# B&R Automation Studio project PLC code - cp (part 13)

### Dryer.typ
```iecst
TYPE
	DryerModel_enum :
		(
		DryerNoType,
		DryerType_NOZ2_NIR_ARCLAMP,
		DryerType_NOZ2_NIR
		);
	DryerMachineStatus_enum :
		(
		DRYERMACH_STOPPED,
		DRYERMACH_PREPARINGTOMOVE,
		DRYERMACH_MOVING,
		DRYERMACH_PREPARING,
		DRYERMACH_PREPARED,
		DRYERMACH_STARTING,
		DRYERMACH_DRYING,
		DRYERMACH_STOPPING_DRYING,
		DRYERMACH_STOPPING_TRANSPORT,
		DRYERMACH_PREPARINGEMPTYBELT, (*Only vaccum transport on*)
		DRYERMACH_ERROR
		);
	Dryer_ProductDetectInputs : 	STRUCT
		pPDSignalSensorL1 : UDINT; (*Pointer to ProductDetect Signal coming directly from the sensor*)
		pPDSignalSensorL2 : UDINT; (*Pointer to ProductDetect Signal coming directly from the sensor*)
	END_STRUCT;
	Dryer_TempInputs : 	STRUCT
		iBoardInRaw : INT;
		iBoardOutRaw : INT;
		iBeltRaw : INT;
		iAirBlowerInputRaw : INT; (*45214336. -50C to +200C. 4-20mA*)
		iAirBlowerOutputRaw : INT; (*45214336. -50C to +200C. 4-20mA*)
		xBoardInSensorError : BOOL; (*Sensor Error*)
		xBoardOutSensorError : BOOL; (*Sensor Error*)
		xBeltSensorError : BOOL; (*Sensor Error*)
		xAirBlowerInputSensorError : BOOL; (*45214336. -50C to +200C. 4-20mA. Sensor Error*)
		xAirBlowerOutputSensorError : BOOL; (*45214336. -50C to +200C. 4-20mA. Sensor Error*)
	END_STRUCT;
	Dryer_InputsButtons : 	STRUCT
		xStopBlowers : BOOL;
		xManual : BOOL;
		xZero : BOOL;
		xAuto : BOOL;
		xStop : BOOL; (*EDGE*)
		xReset : BOOL;
	END_STRUCT;
	Dryer_SafetyInputs : 	STRUCT
		xMovementsEnabled : BOOL;
		xRemoteEStopOK : BOOL; (*Remote Emergency Stop*)
		xEStopFrontOK : BOOL;
		xEStopRearOK : BOOL;
		xClosedFrontInput : BOOL; (*Closed door detection*)
		xClosedFrontOutput : BOOL; (*Closed door detection*)
		xClosedRearInput : BOOL; (*Closed door detection*)
		xClosedRearOutput : BOOL; (*Closed door detection*)
	END_STRUCT;
	Dryer_Inputs : 	STRUCT
		Sw : Dryer_Inputs_Sw;
		Safety : Dryer_SafetyInputs;
		xStart : {REDUND_UNREPLICABLE} BOOL; (*EDGE*)
		xManual_GI : BOOL;
		xZero_GI : BOOL;
		xAuto_GI : BOOL;
		xMute : BOOL;
		xMain24VdcOK : BOOL;
		xFan24VdcOK : BOOL;
		xFanBreakersOK : BOOL;
		xFanBreakersWarning : BOOL; (*Power higher than 80% for all fans*)
		xConsentOk : BOOL;
		xExternalCleaningOrder : BOOL;
		iMachineModelCode : INT;
		xOpenDoorsKey : BOOL; (*Enable open doors with ArcLamp hot*)
		Temp : Dryer_TempInputs;
		ProductDetect : Dryer_ProductDetectInputs;
		Buttons : Dryer_InputsButtons;
	END_STRUCT;
	Dryer_HwData : 	STRUCT
		Family : USINT;
		Name : STRING[20];
		SerialNumber : STRING[80]; (*Serial number of the machine*)
	END_STRUCT;
	Dryer_Excutions : 	STRUCT
		slow : UDINT;
		fast : UDINT;
	END_STRUCT;
	Dryer_States_Position : 	STRUCT
		xGoingToPrint : BOOL; (*Internal bool used on printer to set state NOT CAP/NOT PRINT in printer*)
		xInPrint : BOOL; (*Internal bool used on printer to set state PRINTING in printer*)
		xCleaning : BOOL; (*Internal bool used on printer to set state CLEANING in printer*)
		xGoingToCap : BOOL; (*Internal bool used on printer to set state NOT CAP/NOT PRINT in printer*)
		xInCap : BOOL; (*Internal bool used on printer to set state CAPPED in printer*)
	END_STRUCT;
	Dryer_States_AutoLocation : 	STRUCT
		xLocalORManual : BOOL; (*Local settings and orders*)
		xLocal : BOOL; (*Local settings and orders*)
		xRemote : BOOL; (*Remote settings and orders*)
	END_STRUCT;
	Dryer_States_Mode : 	STRUCT
		xManual : {REDUND_UNREPLICABLE} BOOL; (*State to define Manual Mode*)
		xZero : BOOL; (*State to define Zero Mode*)
		xAuto : BOOL; (*State to define Auto Mode*)
		xStartUp : BOOL; (*State to define StartUp Mode*)
	END_STRUCT;
	Dryer_States_Out : 	STRUCT
		xOnline : BOOL;
		xError : BOOL;
		xDrying : BOOL;
		xDryerPresent : BOOL;
		xReadyToDry : BOOL;
		xJamDetection : BOOL;
		xTransportMoving : BOOL;
		xInRemote : BOOL;
		iModelVersion1 : UINT;
		iModelVersion2 : UINT;
		xMediaPresent : BOOL;
		xReadyToEmptyBelt : BOOL;
		xBeltEmpty : BOOL; (*Belt empty in the device*)
	END_STRUCT;
	Dryer_States_Temp : 	STRUCT
		rBoardIn : REAL;
		rBoardOut : REAL;
		rBelt : REAL;
		rAirBlowerInput : REAL;
		rAirBlowerOutput : REAL;
	END_STRUCT;
	Dryer_States_HMI : 	STRUCT
		xDryerLocalStopped : BOOL;
		xDryerStopped : BOOL;
		xShowThickness : BOOL; (*Thickness and Gap is used in the program and can be adjusted*)
		xVirtualMedia : BOOL;
		xShowEnableNIR : BOOL; (*Variable to let NIR enabling*)
	END_STRUCT;
	Dryer_States : 	STRUCT
		Position : Dryer_States_Position;
		Mode : Dryer_States_Mode;
		AutoLocation : Dryer_States_AutoLocation;
		LocationControl : MachineAutoLocation_enum;
		Out : Dryer_States_Out;
		DryerState : DryerMachineStatus_enum;
		Temp : Dryer_States_Temp;
		xConsent : BOOL; (*Internal bool used on printer to set state in CONSENT printer*)
		iAutoModeSW : INT; (*Printer State to sw *)
		iMachineModelCodeSW : INT; (*Printer model to Sw, in function of HW ID code*)
		xNotAutoPossible : BOOL; (*Some condition is preventing to entering auto*)
		StateMode : enumEFI_GenMachineState; (*states*)
		AutoMode : stEFI_MachineAutoModes; (*commands*)
		uiLicenseCounter : UINT;
		exec : Dryer_Excutions;
		HwData : Dryer_HwData;
		xAnyProductDetect : BOOL; (*Any product detect. In any line and coming from Carriage or Sensor directly. It means that a media has been printed*)
		xProductDetectL1 : BOOL; (*Any product detect in L1. In any line and coming from Carriage or Sensor directly. It means that a media has been printed*)
		xProductDetectL2 : BOOL; (*Any product detect in L2. In any line and coming from Carriage or Sensor directly. It means that a media has been printed*)
		xMediaDetected : BOOL; (*Media detected before product detect. Detected in Analog or in 3sensors*)
		iJamDevices : USINT := 0; (*Quantity of Jam Devices installed in the machine*)
		xStarted : BOOL; (*TRUE if the PLC is running*)
		HMI : Dryer_States_HMI;
	END_STRUCT;
	Dryer_ConstantParameters : 	STRUCT
		rMinThicknessMedia : REAL; (*mm*)
		rMaxThicknessMedia : REAL; (*mm*)
		rMountedMediaLevelInBypassMode : REAL; (*mm*)
		rMinMargin : REAL; (*mm*)
		rMaxMargin : REAL; (*mm*)
		rDistanceThicknesToPD : REAL; (*Distance Between Thicknes Detection To PD Sensor (mm)*)
		iNumBlocks : USINT; (*For writting the number of blocks in a machine*)
		iNumTransVacuum : USINT; (*For writting the number of TransportVacuum in a machine*)
		iNumJamModules : USINT; (*DEPRECATED!!. //TODELETE For writing the number of Jam Detection modules in a machine*)
		iNumSensorsPerJamDevice : USINT := 4; (*For writing the number of Sensors in each Jam Device*)
		rMaxBeltTorque : REAL := 25; (*Max torque supported by the Belt, independently of the motor itself in N·m*)
		rMaxBeltTempSlow : REAL := 180; (*Max temperature supported by the Belt during 30sec, in ºC*)
		rMaxBeltTempFast : REAL := 190; (*Max temperature supported by the Belt during 2sec, in ºC*)
	END_STRUCT;
	Dryer_CleanBeltParameters : 	STRUCT
		xCleanBeltContinue : BOOL; (*Input software parameter from Sw*)
		xCleanBeltByTiles : BOOL; (*Input software parameter from Sw*)
		xCleanBeltByTime : BOOL; (*Input sw param using time param iCleaningBeltByTime*)
		tiCleaningBeltDuration : TIME; (*Time in seconds. Input software parameter from Sw*)
		iCleaningBeltByTime : UINT; (*Time in Minutes. Input software parameter from Sw*)
		xCleanBeltForced : BOOL; (*Edge Command. Input software parameter from Sw*)
		iSPTilesToCleanBelt : UINT; (*Input software parameter from Sw*)
	END_STRUCT;
	Dryer_SuctionParameters : 	STRUCT
		iBlowerMode : INT; (*Suction mode functionality. It can be configured by GUI with Ventrui when is 1 or Turbine when is 2. Parameters received from GUI*)
		tiBlowerDelayOff : TIME; (*Delay time before turning off the turbine in auto mode*)
	END_STRUCT;
	Dryer_SafetyParameters : 	STRUCT
		rMarginSafePrint : REAL; (*SoftwareInput. Fix offset to bent tile. The heads go to the thickness measured + this value. Value in mm*)
		rMaxBeltSpeedSetPoint : REAL := 70.0; (*Max speed received from gui in m/min*)
	END_STRUCT;
	Dryer_DocumentParameters : 	STRUCT
		rWidth : REAL; (*Board's width in mm*)
		rLength : REAL; (*Board's length in mm*)
		rOffsetL1 : REAL;
		rOffsetL2 : REAL;
	END_STRUCT;
	Dryer_ThermalInertiaReduction : 	STRUCT
		iBoardsToStartReducing : USINT; (*Total boards detected to start reducing the power*)
		iBoardsToMaxPowerReduction : USINT; (*Total boards detected to form maximum power reduction*)
		rMaxPowerReduction : REAL; (*Maximum power reduction for thermal inertia*)
	END_STRUCT;
	Dryer_MediaParameters : 	STRUCT
		rThickness : REAL; (*Tile thickness to print from gui in mm*)
		rWidth : REAL; (*Board's width in mm*)
		rGap : REAL; (*Gap between boards in mm*)
		rLength : REAL; (*Board's length in mm*)
		rMargin : REAL; (*SoftwareInput, dry margin in mm*)
		rOffsetRegisterL1 : REAL;
	END_STRUCT;
	Dryer_SwParameters : 	STRUCT
		CleanBelt : Dryer_CleanBeltParameters;
		Suction : Dryer_SuctionParameters;
		Safety : Dryer_SafetyParameters;
		Media : stThicknessCtrl_MediaConfig;
		xDoubleLine : BOOL; (*0: Derecha 1: Izquierda*)
		xMachineDirection : BOOL; (*0: Derecha 1: Izquierda*)
		xEnableNir : BOOL;
		xEnableDDC : BOOL; (*Enable DDC in Dryer*)
		xEnableArcLamp : BOOL;
		rSubstratePowerReduction : REAL := 1.0; (*Substrate power reduction. From 1.0 (default) to 0.3 is allowed*)
		tiDelayConsent : TIME; (*Used on kernel to PLC. Time in seconds*)
		rBeltSpeedSetPoint : REAL := 20.0; (*Speed in m/min. Input parameter from SW*)
		xLineEmptyingBelt : BOOL; (*Line in emptying belt*)
		xPrinterBeltRuning : BOOL; (*Printer belt runing status*)
	END_STRUCT;
	Dryer_Parameters : 	STRUCT
		SW : Dryer_SwParameters; (*Software input params*)
		CT : Dryer_ConstantParameters; (*Printer input constants params*)
		ThermalInertia : Dryer_ThermalInertiaReduction;
		ConfigName : STRING[80];
		ConfigNameID : USINT := 0; (*Identification of the Configuration been executed*)
		xTransVacuumIndependenParams : BOOL; (*TRUE: Each TransVacuum with different parameters. FALSE: TransVacuum[1] copied to the rest of elements*)
		MachineModel : DryerModel_enum; (*HW ID codes are defined here*)
		PDSignalTpe : ProductDetectSignal_enum;
		xLeftHandMachine : BOOL; (*Software Output*)
		xRightHandMachine : BOOL; (*Software Output*)
		xLocalDisableDDC : BOOL;
		xEnableDryDocWidth : BOOL; (*Enable drying width by image instead of media, only in remote mode.*)
	END_STRUCT;
	Dryer_commands_Auto : 	STRUCT
		xPrepareToDry : BOOL;
		xStartDrying : BOOL;
		xRunTransport : BOOL;
		xPrepareToEmptyBelt : BOOL;
	END_STRUCT;
	Dryer_commands : 	STRUCT
		xAllToCap : BOOL; (*Use as EDGE*)
		xAllToPrint : BOOL; (*Use as EDGE*)
		xToLocal : BOOL; (*Command to go in Local mode*)
		xToRemote : BOOL; (*Command to go in Remote mode*)
		xResetSwitch : BOOL;
		xResetHub : BOOL;
		xResetFanBreaker : BOOL;
		xUnlockDoors : BOOL; (*Use as EDGE*)
		SerialNumber : stGeneral_SerialNumberCommands;
	END_STRUCT;
	Dryer_Inputs_Sw : 	STRUCT
		xStart_GI : BOOL; (*EDGE*)
		xStop_GI : BOOL; (*Edge command*)
		xMute_GI : BOOL; (*EDGE*)
		xPause_GI : BOOL; (*EDGE*)
		xReset_GI : BOOL; (*EDGE*)
		xToStop_GI : BOOL; (*Edge commandBool to Stop Mode*)
		xToNormal_GI : {REDUND_UNREPLICABLE} BOOL; (*Edge commandBool to start AutoRun Mode*)
		xToByPass_GI : BOOL; (*Edge commandBool to start Bypass Mode*)
		xStopBlowers_GI : BOOL; (*To stop blowers after keep them off to avoid cardboard fire*)
	END_STRUCT;
	Dryer_AutoCommands : 	STRUCT
		iAutoMode : enumEFI_MachineAutoStatesMode; (*Internal variable to manage AUTOMATIC modes in printer RU,BUPASS, LAB AND STOP*)
		xMuteAlarms : BOOL; (*Edge commandBool used to mute all alarms*)
		xToCap : BOOL; (*Edge commandBool used to send all block to cap*)
		xToPrint : BOOL; (*Edge commandBool used to send all block to print*)
		xReset : BOOL; (*Internal bool used on printer to set state RESET in printer*)
		xStart : BOOL; (*Edge Command to Start the Machine. By button or an specific order from Sw*)
		xStop : BOOL; (*Edge Command to Stop the Machine. By button or an specific order from Sw*)
	END_STRUCT;
	Dryer_AlarmsSafety : 	STRUCT
		xMaintenanceKey : BOOL; (*Maintenance Key active. Enables without safety guard closed*)
		xRemoteEStop : BOOL; (*Remote Emergency Stop*)
		xEStopFront : BOOL; (*Emergency Stop*)
		xEStopRear : BOOL; (*Emergency Stop*)
		xOpenedFrontInput : BOOL; (*Door*)
		xOpenedFrontOutput : BOOL; (*Door*)
		xOpenedRearInput : BOOL; (*Door*)
		xOpenedRearOutput : BOOL; (*Door*)
	END_STRUCT;
	Dryer_AlarmsList : 	STRUCT
		Safety : Dryer_AlarmsSafety;
		xAlarmPlarformInc : BOOL; (*AlarmCritical*)
		xAlarmComPcPLC : BOOL; (*AlarmStop*)
		xAlarmMountedMedia : BOOL;
		xAlarmMountedPieceBypassMode : BOOL; (*AlarmStop*)
		xUpNotConsent : BOOL; (*Resume alarms*)
		xNoActionDangerCollision : BOOL; (*Resume alarms*)
		xNoActionAlarmExist : BOOL; (*Resume alarms*)
		xPDBrokenSensorL1 : BOOL; (*Product Detect Line 1 Broken or Desconected*)
		xPDBrokenSensorL2 : BOOL; (*Product Detect Line 2 Broken or Desconected*)
		xMain24Vdc : BOOL; (*Main 24VDC Power Supply switched off*)
		xFan24Vdc : BOOL; (*Fan 24VDC Power Supply switched off*)
		xFanBreakers : BOOL; (*Fan breakers error*)
		xAlrBeltOvertorque : BOOL; (*Alarm Critical: Overtorque in Belt. Risk to break the belt itself*)
		xAlrBeltOverTempSlow : BOOL; (*Alarm Critical: OverTemperature in Belt. Risk to break the belt itself*)
		xAlrBeltOverTempFast : BOOL; (*Alarm Critical: OverTemperature in Belt. Risk to break the belt itself*)
		xAlrJam : BOOL; (*Alarm Critical: Any jam is triggered*)
		xAlrWrongPhysConf : BOOL; (*Alarm Critical: Wrong physical configuration or some tarjet are disconected*)
	END_STRUCT;
	Dryer_WarningsList : 	STRUCT
		xNotEnabledMovement : BOOL;
		xKeyMantenanceActive : BOOL; (*Key mantenance is active. No movements*)
		xValidConfiguration : BOOL; (*Review*)
		xMaxMovsBentTile : BOOL;
		xBentMedia : BOOL;
		xFanBreakersHighLoad : BOOL; (*Fan breakers High Load*)
		xMountedMediaInside : BOOL;
		xMediaStoppedInside : BOOL;
		xBoardInSensorError : BOOL; (*Sensor Error*)
		xBoardOutSensorError : BOOL; (*Sensor Error*)
		xBeltSensorError : BOOL; (*Sensor Error*)
		xAirBlowerInputSensorError : BOOL; (*45214336. -50C to +200C. 4-20mA. Sensor Error*)
		xAirBlowerOutputSensorError : BOOL; (*45214336. -50C to +200C. 4-20mA. Sensor Error*)
		xFrontDoorOpened : BOOL;
		xJamLowCrash : BOOL; (*Low level jam detected by the jam device*)
		xRearDoorOpened : BOOL;
	END_STRUCT;
	Dryer_Alarms : 	STRUCT
		Warning : Dryer_WarningsList;
		Alarm : Dryer_AlarmsList;
		xAlrStopDrying : BOOL;
		iReasonStopDrying : UINT;
		xAlrDisableGoToProduction : BOOL;
		xAlrSafetySystemEStop : BOOL; (*SLX DI 10 is enable transport from safety progam*)
		xAlarmSound : BOOL;
	END_STRUCT;
	Dryer_Log : 	STRUCT
		ManualChg : DINT;
		AutoChg : DINT;
		ManualHrs : DINT;
		AutoHrs : DINT;
		VdcHrs : DINT;
		DateStart : DINT;
		iPieceCounterBtwCleaningsL2 : INT;
		iPieceCounterBtwCleaningsL1 : INT;
		udiBentTilesCounter : UDINT;
		udiPiecesCounterErrorL1 : UDINT; (*PD Detection Counter Failed L1*)
		udiPiecesCounterErrorL2 : UDINT; (*PD Detection Counter Failed L2*)
		udiPiecesCounterL1 : UDINT;
		udiPiecesCounterL2 : UDINT;
		udiTileCounterBalluffLaser : UDINT; (*Program in mode active..end*)
		udiTileCounterTriggerLaser : UDINT; (*Program in mode active..end*)
		udiDifCounters : UDINT; (*Program in mode active..end*)
		iTilesCounterToClean : UINT;
	END_STRUCT;
	Dryer_Outputs : 	STRUCT
		xResetSwitch : BOOL;
		xResetHub : BOOL;
		xResetFanBreaker : BOOL;
		xLockFrontDoor : BOOL;
		xLockRearDoor : BOOL;
		xBuzzer : BOOL;
		xRedLight : BOOL;
		xYellowLight : BOOL;
		xBlueLight : BOOL;
		xWhiteLight : BOOL;
		xResetBlueLight : BOOL;
		xConsentL1 : BOOL;
		xConsentL2 : BOOL;
		xSuctionTurbine : BOOL;
		xLightReset : BOOL;
		xCoolingPCStart : BOOL;
		xKeepSafetyNIR : BOOL;
	END_STRUCT;
	DryerMachine : 	STRUCT
		In : Dryer_Inputs;
		St : Dryer_States;
		Pt : Dryer_Parameters;
		commands : Dryer_commands;
		AutoCmd : Dryer_AutoCommands;
		AlSummary : stEFI_AlarmSummary;
		Al : Dryer_Alarms;
		Lg : Dryer_Log;
		Out : Dryer_Outputs;
	END_STRUCT;
	DryerRemoteSignals : 	STRUCT
		xMediaPresent : BOOL; (*Media present at the entrance of the machine*)
		xBreakerOKBlowerInput : BOOL;
		xBreakerOKBlowerOutput : BOOL;
		Safety : Dryer_SafetyInputs;
	END_STRUCT;
	DryerRemoteData : 	STRUCT
		xCommsOK : BOOL; (*The comunications are working fine. Data can be trusted*)
		Parameters : Dryer_SwParameters;
		Commands : Dryer_commands_Auto; (*From Line to Dryer*)
		Signals : DryerRemoteSignals;
	END_STRUCT;
END_TYPE
```

### InksBox.typ
```iecst
TYPE
	InkboxCabinetParameters : 	STRUCT
		MaxTempPowerPsu : UINT; (*Power in Watts*)
		TotalInksPerPsu : USINT;
		TotalInkSystems : USINT;
	END_STRUCT;
	InkboxParameters : 	STRUCT
		TotalCabinets : USINT;
		Cabinets : ARRAY[0..MAX_LAST_INK_CABINET]OF InkboxCabinetParameters;
	END_STRUCT;
	InkboxCabinetStatus : 	STRUCT
		xExists : BOOL; (*The cabinet exists*)
		rPowerReduction : REAL; (*Power reduction calculated*)
		rTotalAskedPower : REAL; (*The total power calculated by the Inks*)
	END_STRUCT;
	InkboxCommands : 	STRUCT  (*Just Edge commands*)
		xReset : BOOL;
		xMute : BOOL;
	END_STRUCT;
	InkboxStatus : 	STRUCT
		iTotalInks : USINT; (*Total possible Inks by cabinets configuration*)
		ExistingInks : ARRAY[0..MAX_LAST_INK]OF BOOL;
		Cabinets : ARRAY[0..MAX_LAST_INK_CABINET]OF InkboxCabinetStatus;
	END_STRUCT;
	InkBox : 	STRUCT
		Status : InkboxStatus;
		Parameters : InkboxParameters;
		Commands : InkboxCommands; (*Just Edge Commands*)
	END_STRUCT;
END_TYPE
```

### Global.var
```iecst
VAR
	iIndexWhiteCuringLedBar : USINT;
	iIndexColorCuringLedBar : USINT;
	iIndexPrimerCuringLedBar : USINT;
	gSafetyController : stSafetyController;
	gBelt : stBelt;
	gBeltClean : BeltClean_typ;
	gBlock : ARRAY[0..MAX_LAST_BLOCK] OF StBlock; (*Logical array of Blocks in the machine. Starts in 0 because it is used in a C program*)
	gSimpleBlock : ARRAY[0..MAX_LAST_SIMPLEBLOCK] OF SimpleBlock; (*Logical array of Blocks in the machine. Starts in 0 because it is used in a C program*)
	gBlockInputs : ARRAY[0..MAX_LAST_BLOCK] OF StBlock_Inputs; (*Used for mapping physical inputs block to logical block*)
	gBlockOutputs : ARRAY[0..MAX_LAST_BLOCK] OF StBlock_Outputs; (*Used for mapping physical outputs block to logical block*)
	gPowermeters : ARRAY[0..2] OF stPowerMeter;
	gChiller : ARRAY[0..MAX_LAST_CHILLER] OF StChiller; (*Struct for chiller configuration*)
	gPlcDiagMC_Pt : StGeneral_Parameters;
	gTransVacuum : ARRAY[0..MAX_LAST_TRANS_VACUUM] OF TransVacuum_typ;
	gNonCrash : ARRAY[0..MAX_LAST_NON_CRASH] OF NonCrash_typ;
	gCuringLed : ARRAY[0..MAX_LAST_CURING_LED] OF CuringLed_typ;
	gDing : stThicknessAnalog_typ;
	gOverVarnish : Opv_typ;
	gPrimer : Primer_typ;
	gStacker : Stacker_typ;
	gDryerAnc : DryerAnc_typ;
	gLine : LineControl_typ;
	gEventLogLoader : EventLoader;
	gEventLogManager : EventManager;
	gInks : ARRAY[0..MAX_LAST_INK] OF stInks; (*Logical array of InkSystems in the machine. Starts in 0 because it is used in a C program*)
	gInksConstants : stInksConstantsToSw; (*horrible!! Pending to change *)
	gSarm : Sarm_typ;
	gFeeder : Feeder_typ;
	gInksInputs : ARRAY[0..MAX_LAST_INK] OF stInksSignalsIn; (*0 is not used. Just to compile in C*)
	gInksOutputs : ARRAY[0..MAX_LAST_INK] OF stInksSignalsOut;
	gJamInputs : ARRAY[0..MAX_LAST_JAMDEVICE] OF JamDetectInputs_typ;
	gJamOutputs : ARRAY[0..MAX_LAST_JAMDEVICE] OF JamDetectOutputs_typ;
	gMachine : StGeneral;
	gDryer : DryerMachine;
	gNirAdphos : NIRAdphos;
	gPairedMotors : ARRAY[0..2] OF PairedIclaMotors_typ; (*Paired icla motors structure*)
	gEdgeHoldDown : EdgeHoldDown_typ; (*Edge hold down structure*)
	gPhotoCells : nSensors_typ; (*gPhotocells structure*)
	gPLC : StPLC;
	gThicknessCtrl : stThicknessCtrl_typ;
	gBasicDetectMedia : DetectionMedia;
	gArcLampGew : ArcLampGew;
	g_xInputSelectMachine : BOOL;
	gJamDetect : ARRAY[0..MAX_LAST_JAMDEVICE] OF JamDetect_typ;
	gAirCleaner : StGeneral_AirCleaner;
	gCamera : StGeneral_Camera;
	gJamCamera : JamPerBar_typ;
	gJamPerCuringLed : ARRAY[0..MAX_LAST_CURING_LED] OF JamPerBar_typ;
	gJamPerInk : ARRAY[0..MAX_LAST_INK] OF JamPerBar_typ;
	gInkBox : InkBox;
	gTime : TimeMachine;
	gInverterSignalsPowerLink : ARRAY[0..MAX_LAST_INVERTER] OF AxisP66_Signals_typ;
	gInverterSignalsCanOpen : ARRAY[0..MAX_LAST_INVERTER] OF AxisP66_Signals_typ;
	gInverterSignalsPowerLinkABB : ARRAY[0..MAX_LAST_INVERTER] OF AxisP66_Signals_typ;
	gPlcCards : ARRAY[0..100] OF PLCCardData;
	xShowSecondLayout : BOOL := FALSE; (*Show second card block layout in diagnostic screen*)
	xShowThirdLayout : BOOL := FALSE; (*Show third card block layout in diagnostic screen*)
	stConfigToShow_Lyout1 : STRING[80] := 'P4_PDC_content'; (* Configuration ID to show in HMI || P4_PDC_content ; SHIELD_Cards_content ; NZ2_Cards_content*)
	stConfigToShow_Lyout2 : STRING[80] := 'P4_block1_content'; (*Configuration ID to show in HMI || P4_block1_content ; NZ2_Printer_content*)
	stConfigToShow_Lyout3 : STRING[80] := 'P4_block2_content'; (*Configuration ID to show in HMI || P4_block2_content*)
END_VAR
```

### Global_IO.var
```iecst
VAR
	X20CPUData : PlcCardMapping; (*Map: P4&EBRO*)
	X1 : PlcCardMapping; (*Map: P4&EBRO*)
	X2 : PlcCardMapping; (*Map: P4&EBRO*)
	X3 : PlcCardMapping; (*Map: P4&EBRO*)
	X20DOF322_001 : PlcCardMapping; (*Map: P4*)
	X20DIF371_001 : PlcCardMapping; (*Map: EBRO&S1400*)
	X20DIF371_002 : PlcCardMapping; (*Map: P4&EBRO&S1400*)
	X20DIF371_003 : PlcCardMapping; (*Map: P4&EBRO$S1400*)
	X20DOF322_004 : PlcCardMapping; (*Map: P4*)
	X20DIF371_004 : PlcCardMapping; (*Map: EBRO*)
	X20DIF371_005 : PlcCardMapping; (*Map: S1400*)
	X20DIF371_006 : PlcCardMapping; (*Map: S1400*)
	X20AI2636_005 : PlcCardMapping; (*Map: P4*)
	X20DOF322_005 : PlcCardMapping; (*Map: EBRO*)
	X20SLX402_006 : PlcCardMapping; (*	X20SI2100_010 : PlcCardMapping; Map: P4*)
	X20DOF322_006 : PlcCardMapping; (*Map: EBRO*)
	X20AI4322_008 : PlcCardMapping; (*Map: EBRO*)
	X20AI4322_102 : PlcCardMapping; (*Map: InkBox*)
	X20AI4322_202 : PlcCardMapping; (*Map: InkBox*)
	X20AI4322_302 : PlcCardMapping; (*Map: InkBox*)
	X20AT2222_103 : PlcCardMapping; (*Map: InkBox*)
	X20AT2222_203 : PlcCardMapping; (*Map: InkBox*)
	X20AT2222_303 : PlcCardMapping; (*Map: InkBox*)
	X20DOF322_104 : PlcCardMapping; (*Map: InkBox*)
	X20DOF322_204 : PlcCardMapping; (*Map: InkBox*)
	X20DOF322_304 : PlcCardMapping; (*Map: InkBox*)
	X20AO4622_105 : PlcCardMapping; (*Map: InkBox*)
	X20AO4622_205 : PlcCardMapping; (*Map: InkBox*)
	X20AO4622_305 : PlcCardMapping; (*Map: InkBox*)
	X20DI9372_008 : PlcCardMapping; (*Map: S1400*)
	X20AO4622_009 : PlcCardMapping; (*Map: EBRO*)
	X20DOF322_009 : PlcCardMapping; (*Map:S1400*)
	X20DOF322_010 : PlcCardMapping; (*Map:S1400*)
	X20AT4222_010 : PlcCardMapping; (*Map: EBRO*)
	X20DOF322_011 : PlcCardMapping; (*Map:S1400*)
	X20DOF322_012 : PlcCardMapping; (*Map:S1400*)
	X20DOF322_013 : PlcCardMapping; (*Map:S1400*)
	X20AI8321_015 : PlcCardMapping; (*Map:S1400*)
	X20AI8321_016 : PlcCardMapping; (*Map:S1400*)
	X20AI8321_111 : PlcCardMapping; (*Map:S1400*)
	X20AI8321_112 : PlcCardMapping; (*Map:S1400*)
	X20AI8321_113 : PlcCardMapping; (*Map:S1400*)
	X20AI8321_114 : PlcCardMapping; (*Map:S1400*)
	X20AI8321_018 : PlcCardMapping; (*Map:S1400*)
	X20AI8321_019 : PlcCardMapping; (*Map:S1400*)
	X20AO4622_017 : PlcCardMapping; (*Map:S1400*)
	X20AO4622_018 : PlcCardMapping; (*Map:S1400*)
	X20AO4622_019 : PlcCardMapping; (*Map:S1400*)
	X20AO4622_020 : PlcCardMapping; (*Map:S1400*)
	X20AT4222_022 : PlcCardMapping; (*Map:S1400*)
	X20AT4222_023 : PlcCardMapping; (*Map:S1400*)
	X20AI2636_024 : PlcCardMapping; (*Map:S1400*)
	X20AI8321_025 : PlcCardMapping;
	X20AI8321_024 : PlcCardMapping;
	X20DIF371_024 : PlcCardMapping; (*Map:S1400*)
	X20AI8321_026 : PlcCardMapping; (*Map:S1400*)
	X20AT4222_027 : PlcCardMapping;
	X20AT4222_028 : PlcCardMapping;
	X20AT4222_029 : PlcCardMapping; (*Map:S1400*)
	X20AT4222_030 : PlcCardMapping; (*Map:S1400*)
	X20DIF371_030 : PlcCardMapping; (*Map: P4*)
	X20AI2636_100 : PlcCardMapping;
	X20DIF371_101 : PlcCardMapping; (*Map: P4 & Map: InkBox*)
	X20DIF371_102 : PlcCardMapping; (*Map: P4*)
	X20DIF371_103 : PlcCardMapping; (*Map: P4*)
	X20DIF371_104 : PlcCardMapping; (*Map: P4*)
	X20DIF371_105 : PlcCardMapping; (*Map: P4*)
	X20DIF371_106 : PlcCardMapping; (*Map: P4*)
	X20DI9372_107 : PlcCardMapping; (*Map: P4*)
	X20DIF371_107 : PlcCardMapping; (*Map: P4*)
	X20DC4395_104 : PlcCardMapping; (*Map: P4*)
	X20DC4395_105 : PlcCardMapping; (*Map: P4*)
	X20DOF322_106 : PlcCardMapping; (*Map: P4*)
	X20DOF322_107 : PlcCardMapping; (*Map: P4*)
	X20DOF322_108 : PlcCardMapping; (*Map: P4*)
	X20DOF322_109 : PlcCardMapping; (*Map: P4*)
	X20DOF322_110 : PlcCardMapping; (*Map: P4*)
	X20AI8321_109 : PlcCardMapping; (*Map: P4*)
	X20AI8321_110 : PlcCardMapping; (*Map: P4*)
	X20AO4622_111 : PlcCardMapping; (*Map: P4*)
	X20AO4622_112 : PlcCardMapping; (*Map: P4*)
	X20AO4622_113 : PlcCardMapping; (*Map: P4*)
	X20AO4622_114 : PlcCardMapping; (*Map: P4*)
	X20AO4622_115 : PlcCardMapping; (*Map: P4*)
	X20AO4622_116 : PlcCardMapping; (*Map: P4*)
	X20AO4622_117 : PlcCardMapping; (*Map: P4*)
	X20AT4222_114 : PlcCardMapping; (*Map: P4*)
	X20AT4222_115 : PlcCardMapping; (*Map: P4*)
	X20AT4222_116 : PlcCardMapping; (*Map: P4*)
	X20AT4222_117 : PlcCardMapping; (*Map: P4*)
	X20AT4222_118 : PlcCardMapping; (*Map: P4*)
	X20AT4222_119 : PlcCardMapping; (*Map: P4*)
	X20AT4222_120 : PlcCardMapping; (*Map: P4*)
	X20AT4222_121 : PlcCardMapping; (*Map: P4*)
	X20CS1030_150 : PlcCardMapping; (*Map: P4*)
	X20CS1030_151 : PlcCardMapping; (*Map: P4*)
	X20CS1030_121 : PlcCardMapping; (*Map: P4*)
	X20CS1030_180 : PlcCardMapping; (*Map: P4*)
	X20CS1030_181 : PlcCardMapping; (*Map: P4*)
	X20CS1030_162 : PlcCardMapping; (*Map: P4*)
	X20PS3300_114 : PlcCardMapping; (*Map: P4*)
	Pdc_X20DOF322_024 : PlcCardMapping;
	Pdc_X20DOF322_025 : PlcCardMapping;
	Pdc_X20DIF371_023 : PlcCardMapping;
	X20PS3300_106 : PlcCardMapping; (*Map: P4*)
	X20PS3300_020 : PlcCardMapping;
	X20PS3300_008 : PlcCardMapping;
	X20PS3300_157 : PlcCardMapping;
	X20PS3300_150 : PlcCardMapping;
	X20PS3300_115 : PlcCardMapping;
	X20PS3300_107 : PlcCardMapping;
	X20PS3300_152 : PlcCardMapping; (*Map: P4*)
	X20DIF371_151 : PlcCardMapping; (*Map: P4*)
	X20DIF371_152 : PlcCardMapping; (*Map: P4*)
	X20DIF371_153 : PlcCardMapping; (*Map: P4*)
	X20DIF371_154 : PlcCardMapping; (*Map: P4*)
	X20DOF322_155 : PlcCardMapping; (*Map: P4*)
	X20DOF322_156 : PlcCardMapping; (*Map: P4*)
	X20AI8221_156 : PlcCardMapping; (*Map: P4*)
	X20AO4622_157 : PlcCardMapping; (*Map: P4*)
	X20AO4622_158 : PlcCardMapping; (*Map: P4*)
	X20AO4622_159 : PlcCardMapping; (*Map: P4*)
	X20AO4622_160 : PlcCardMapping; (*Map: P4*)
	X20AO4622_161 : PlcCardMapping; (*Map: P4*)
	X20SI8110_117 : PlcCardMapping; (*Map: P4*)
	X20SO2110_118 : PlcCardMapping; (*Map: P4*)
	X20DIF371_201 : PlcCardMapping; (*Map: P4 & InkBox*)
	X20DIF371_202 : PlcCardMapping; (*Map: P4*)
	X20DIF371_203 : PlcCardMapping; (*Map: P4*)
	X20DIF371_301 : PlcCardMapping; (*Map: InkBox*)
	X20DC4395_204 : PlcCardMapping; (*Map: P4*)
	X20DC4395_205 : PlcCardMapping; (*Map: P4*)
	X20DIF371_180 : PlcCardMapping; (*Map: P4*)
	X20AI8321_181 : PlcCardMapping; (*Map: P4*)
	X20DOF322_205 : PlcCardMapping; (*Map: Dryer*)
	X20DOF322_206 : PlcCardMapping; (*Map: P4*)
	X20DOF322_207 : PlcCardMapping; (*Map: P4*)
	X20DOF322_208 : PlcCardMapping; (*Map: P4*)
	X20AI8321_207 : PlcCardMapping; (*Map: P4*)
	X20AI8321_209 : PlcCardMapping; (*Map: P4*)
	X20AI8321_210 : PlcCardMapping; (*Map: P4*)
	X20AO4622_208 : PlcCardMapping; (*Map: Dryer*)
	X20AO4622_211 : PlcCardMapping; (*Map: P4*)
	X20AO4622_212 : PlcCardMapping; (*Map: P4*)
	X20AO4622_213 : PlcCardMapping; (*Map: P4*)
	X20AT4222_209 : PlcCardMapping; (*Map: Dryer*)
	X20AT4222_214 : PlcCardMapping; (*Map: P4*)
	X20AT4222_215 : PlcCardMapping; (*Map: P4*)
	X20AT4222_216 : PlcCardMapping; (*Map: P4*)
	X20SI8110_217 : PlcCardMapping; (*Map: P4*)
	X20SO2110_218 : PlcCardMapping; (*Map: P4*)
	Reserve01 : PlcCardMapping;
	SiUnitBK1 : StSiUnit;
	SiUnitBK2 : StSiUnit;
	SiUnitPwrLnkBK1 : StSiUnitPwrLnk;
	Pdc_X20DIF371_001 : PlcCardMapping;
	Pdc_X20DIF371_002 : PlcCardMapping;
	Pdc_X20DIF371_003 : PlcCardMapping;
	Pdc_X20DIF371_004 : PlcCardMapping;
	Pdc_X20DIF371_005 : PlcCardMapping;
	Pdc_X20DIF371_006 : PlcCardMapping;
	Pdc_X20DIF371_007 : PlcCardMapping;
	Pdc_X20DIF371_009 : PlcCardMapping;
	Pdc_X20DIF371_030 : PlcCardMapping;
	Pdc_X20AI2636_050 : PlcCardMapping;
	Pdc_X20DIF371_060 : PlcCardMapping;
	Pdc_X20DIF371_070 : PlcCardMapping;
	X20PS3300_007 : PlcCardMapping;
	Pdc_X20DIF371_024 : PlcCardMapping;
	Pdc_X20DIF371_022 : PlcCardMapping;
	Pdc_X20DIF371_020 : PlcCardMapping;
	Pdc_X20DIF371_021 : PlcCardMapping;
	X20PS3300_006 : PlcCardMapping;
	X20PS3300_022 : PlcCardMapping;
	Pdc_X20DOF322_023 : PlcCardMapping;
	Pdc_X20DIF371_1 : PlcCardMapping;
	Pdc_X20DIF371_2 : PlcCardMapping;
	Pdc_X20DIF371_3 : PlcCardMapping;
	Pdc_X20DOF322_008 : PlcCardMapping;
	Pdc_X20DOF322_009 : PlcCardMapping;
	Pdc_X20DOF322_010 : PlcCardMapping;
	Pdc_X20DOF322_1 : PlcCardMapping;
	Pdc_X20DIF371_050 : PlcCardMapping;
	Pdc_X20DIF371_040 : PlcCardMapping;
	Pdc_X20DOF322_051 : PlcCardMapping;
	Pdc_X20DOF322_011 : PlcCardMapping;
	Pdc_X20DOF322_007 : PlcCardMapping;
	Pdc_X20DOF322_005 : PlcCardMapping;
	X20AO4622_119 : PlcCardMapping;
	X20AO4622_118 : PlcCardMapping;
	X20IF1072_SS1 : PlcCardMapping;
	X20IF1072_SS2 : PlcCardMapping;
	X20IF1072_SS3 : PlcCardMapping;
	X20SM1436_007 : PlcCardMapping;
	X20SM1436_008 : PlcCardMapping;
	X20SM1436_011 : PlcCardMapping;
	X20SM1436_012 : PlcCardMapping;
	X20SM1436_111 : PlcCardMapping;
	X20SM1436_112 : PlcCardMapping;
	X20PS3300_014 : PlcCardMapping;
	X20PS3300_021 : PlcCardMapping;
	X20BC0083 : PlcCardMapping;
	X20PS9400 : PlcCardMapping;
	FakeBoolInput : BOOL;
END_VAR
```

### GlobalComms.var
```iecst
VAR
	gToWriteDataModbSarm : ARRAY[1..25] OF UINT;
	gReceivedDataModbSarm : ARRAY[1..25] OF UINT;
	gToWriteDataModbFeeder : ARRAY[1..25] OF UINT;
	gReceivedDataModbFeeder : ARRAY[1..25] OF UINT;
	gToWriteDataModbStacker : ARRAY[1..25] OF UINT;
	gReceivedDataModbStacker : ARRAY[1..25] OF UINT;
	gToWriteDataModbOpv : ARRAY[1..25] OF UINT;
	gReceivedDataModbOpv : ARRAY[1..25] OF UINT;
	gToWriteDataModbPrimer : ARRAY[1..25] OF UINT;
	gReceivedDataModbPrimer : ARRAY[1..25] OF UINT;
	gToWriteDataModbTransport : ARRAY[1..25] OF INT;
	gReceivedDataModbTransport : ARRAY[1..25] OF INT;
	gReceivedDataModPowerMeter1 : ARRAY[0..120] OF UINT;
	gReceivedDataModPowerMeter2 : ARRAY[0..120] OF UINT;
	gReceivedDataModbSafety : ARRAY[0..20] OF UINT; (*0 Not used. Needed because used in the Tests*)
	gDryerRemoteData : DryerRemoteData; (*This is the data from the Printer to the Dryer*)
	gDryerLocalData : DryerInputs_typ; (*This is the data from the Dryer to the Printer*)
END_VAR
```

### MotionBasis.var
```iecst
(********************************************************************
 * COPYRIGHT - B&R Spain
 ********************************************************************
 * Package: MotionBasis
 * File: MotionBasis.var
 * Author: jorgemur
 * Created: September 19, 2018
 ********************************************************************
 * Variables of Motion
 ********************************************************************)
VAR
	gAxis : ARRAY[0..8] OF AxisCtrl_typ; (*Axis control structure. 1.Belt,2.Bk1,3.Bk2,4.SM1,5.SM2,6.NonCrash1,7.NonCrash28.Bk3*)
END_VAR
VAR RETAIN
	gAxisPermanEncData : ARRAY[0..8] OF MC_ENDLESS_POSITION; (*Permanent variable where encoder data is stored*) (*	gPermanentEncData2 : MC_ENDLESS_POSITION; *) (*Permanent variable where encoder data is stored*)
END_VAR
VAR
	gIcla : ARRAY[0..MAX_LAST_ICLA_MOTOR] OF stIcla; (*Physical array of Icla. index1>>Icla_A index2>>Icla_B*)
	gIclaNetData : ARRAY[0..MAX_LAST_ICLA_MOTOR] OF IclaNetData_typ; (*Physical array of IclaNetData. index1>>Icla_A index2>>Icla_B*)
	gAxisInverter : ARRAY[0..MAX_LAST_INVERTER] OF AxisP66_typ; (*Axis of the Inverters of the system of the family P66 & P67*)
END_VAR
VAR RETAIN
	gISQRippleData : ARRAY[0..8] OF MC_ISQ_RippleData_typ;
END_VAR
(* ********************************************************************
 * Identification of the Axis
 *******************************************************************
 #1. Belt
 #2. Vertical Block 1
 #3. Vertical Block 2
 #4. StepperMotor1 (3 Sensors)
 #5. StepperMotor2 (3 Sensors)
 #6. NonCrash 1
 #7. NonCrash 2
 #8. Vertical Block 3
 ********************************************************************)
```

### Simulation.var
```iecst
VAR
	gSimMachine : SimMachine_typ;
	gSimChiller : ARRAY[0..MAX_LAST_CHILLER] OF stChillerSim;
	gSimBlock : ARRAY[0..MAX_LAST_BLOCK] OF SimBlock_typ;
	gSimSimpleBlock : ARRAY[0..MAX_LAST_SIMPLEBLOCK] OF SimBlock_typ;
	gSimSarm : Sarm_typ;
	gSimFeeder : FeederSim_typ;
	gSimDryerAnc : DryerSimAnc_typ;
	gSimOverVarnish : PrimerSim_typ;
	gSimPrimer : PrimerSim_typ;
	gSimStacker : StackerSim_typ;
	gSimJamDetect : ARRAY[0..MAX_LAST_JAMDEVICE] OF JamDetectSim_typ;
	gSimInks : ARRAY[0..MAX_LAST_INK] OF SimInk_typ;
	gSimSafetyController : SafetyControllerSim_typ;
	gSimArcLamp : ArcLampSim_typ;
	gSimNirAdphos : NirAdphosSim_typ;
	gSimNonCrash : ARRAY[0..MAX_LAST_NON_CRASH] OF SimNonCrash_typ;
	gSimThickCtrl : SimThickCtrl_typ;
	gTestsExec : TestExecution;
	gSimDryer : SimDryer_typ;
END_VAR
```

### Program Logical/InkBox/Config/Initialize (IEC)

#### Initialize.st - Cyclic code
```iecst
PROGRAM _INIT

	HWInfoCpu.pName := ADR(gMachine.St.HwData.Name);
	HWInfoCpu.first := TRUE;
	HWInfoCpu.enable := TRUE;
	HWInfoCpu();
	gMachine.St.HwData.Family := HWInfoCpu.family;

	// Tranfer permanent vars when PLC is starting
	gMachine.parSw:= gPermanentMachine;

	FOR iInksIndex:=1 TO MAX_LAST_INK DO
		gInks[iInksIndex].parSw := gPermanentInksParSw[iInksIndex];
		gInks[iInksIndex].parameters.parBar := gInksPermanentParBar[iInksIndex];
	END_FOR

	gInkBox.Parameters := gPermanentInkBox;
	gBelt.parSw := gPermanentSwBelt;
	gTransVacuum[1].parSw := gPermanentTrVacuum[1];

END_PROGRAM

PROGRAM _CYCLIC

	//Assign the ConfigurationID been executed
	projectInfo(Execute:=gMachine.Pt.ConfigNameID=0); //Just to execute if still the configuration has not been read
	IF projectInfo.Done AND NOT projectInfo.Error THEN
		IF brsstrcmp(ADR(GC_CONFIG_INKBOX),ADR(projectInfo.ConfigurationID))=0 THEN

			IF gMachine.In.x230V THEN //This var is assigned to a ModuleOk just for simulation. Never in a real cabinet
				gMachine.Pt.ConfigNameID:=GC_CONFIG_INKBOX_SIM_ID;
			ELSE
				gMachine.Pt.ConfigNameID:=GC_CONFIG_INKBOX_ID;
			END_IF
		ELSE
			gMachine.Pt.ConfigNameID:=0;
		END_IF
		strcpy(ADR(gMachine.Pt.ConfigName),ADR(projectInfo.ConfigurationID));
	END_IF

END_PROGRAM
```

### Program Logical/InkBox/Config/SavePermanent

#### SavePermanent.st
```iecst
PROGRAM _CYCLIC

	// Permanents Vars
	gPermanentMachine:=gMachine.parSw;

	FOR iInksIndex:=1 TO MAX_LAST_INK DO
		gPermanentInksParSw[iInksIndex] := gInks[iInksIndex].parSw;
		gInksPermanentParBar[iInksIndex] := gInks[iInksIndex].parameters.parBar;
	END_FOR

	gPermanentInkBox := gInkBox.Parameters;
	gPermanentSwBelt := gBelt.parSw;
	gPermanentTrVacuum[1] := gTransVacuum[1].parSw;

	gPermanentVersion.iVersion0 := gPLC.iVersion0;
	gPermanentVersion.iVersion1 := gPLC.iVersion1;
	gPermanentVersion.iVersion2 := gPLC.iVersion2;
	gPermanentVersion.iVersion3 := gPLC.iVersion3;

END_PROGRAM
```

### Program Logical/InkBox/InkBoxCtrl/MainInkBox (IEC)

#### InternalPLC.st - Internal PLC Vars
```iecst
ACTION InternalPLC:

	// PLC VARS
	IF gPLC.diCycleTime =0 THEN
		gPLC.Internal.RestartInfo(enable := TRUE);
		gPLC.diCycleTime:=gPLC.Internal.RestartInfo.cycle_time;  // Is a fix cycle time

		gPLC.xColdRestart:= gPLC.Internal.RestartInfo.init_reason=1;
		gPLC.xWarmRestart:= gPLC.Internal.RestartInfo.init_reason=2;
		gPLC.xDownloadRestart:= gPLC.Internal.RestartInfo.init_reason=3;

		gPLC.xFirst_Scan :=	gPLC.Internal.RestartInfo.init_reason=-1 OR gPLC.xColdRestart OR gPLC.xWarmRestart OR gPLC.xDownloadRestart;

		gPLC.Internal.RestartInfo(enable := FALSE);

	ELSIF gPLC.xFirst_Scan THEN
		gPLC.xFirst_Scan:= FALSE;
		gPLC.xColdRestart:= FALSE;
		gPLC.xWarmRestart:= FALSE;
		gPLC.xDownloadRestart:= FALSE;
	END_IF

	//BLINK
	gPLC.Internal.Blink_100ms.T_Blink:=T#100MS;
	gPLC.Internal.Blink_100ms();
	gPLC.xBlk_100ms:= gPLC.Internal.Blink_100ms.Out;

	gPLC.Internal.Blink_200ms.T_Blink:=T#200MS;
	gPLC.Internal.Blink_200ms();
	gPLC.xBlk_200ms:= gPLC.Internal.Blink_200ms.Out;

	gPLC.Internal.Blink_500ms.T_Blink:=T#500MS;
	gPLC.Internal.Blink_500ms();
	gPLC.xBlk_500ms:= gPLC.Internal.Blink_500ms.Out;

	gPLC.Internal.Blink_1s.T_Blink:=T#1S;
	gPLC.Internal.Blink_1s();
	gPLC.xBlk_1s:= gPLC.Internal.Blink_1s.Out;

	gPLC.Internal.Blink_2s.T_Blink:=T#2S;
	gPLC.Internal.Blink_2s();
	gPLC.xBlk_2s:= gPLC.Internal.Blink_2s.Out;

	gPLC.Internal.Blink_5s.T_Blink:=T#5S;
	gPLC.Internal.Blink_5s();
	gPLC.xBlk_5s:= gPLC.Internal.Blink_5s.Out;

	gPLC.Internal.Blink_10s.T_Blink:=T#10S;
	gPLC.Internal.Blink_10s();
	gPLC.xBlk_10s:= gPLC.Internal.Blink_10s.Out;

	// License counter	and  Keep alive
	IF EDGEPOS(gPLC.xBlk_1s) THEN
		gMachine.St.uiLicenseCounter:= gMachine.St.uiLicenseCounter+1;
		gMachine.St.iFaultRunPlc:= gMachine.St.iFaultRunPlc+1;
	END_IF;

END_ACTION

ACTION resetPLC:

    // Version
	IF gMachine.commands.ResetCpu.AutorizationCode <> 'h98o76' THEN
		RETURN;
	END_IF

	IF EDGEPOS(gMachine.commands.ResetCpu.xExecuteReset) THEN
		statusReset := SYSreset(enable:= TRUE, mode:= 2);
	END_IF

END_ACTION

ACTION setSerialNumber:

    // If the PLC has version, return
	IF brsstrlen(ADR(gMachine.St.HwData.SerialNumber)) > 0 THEN
		RETURN;
	END_IF

	IF EDGEPOS(gMachine.commands.SerialNumber.xExecute) THEN
		brsstrcpy(ADR(gMachine.St.HwData.SerialNumber),ADR(gMachine.commands.SerialNumber.SerialNumber));
		gMachine.commands.SerialNumber.xExecute := FALSE;
	END_IF

END_ACTION
```

#### Calculations.st
```iecst
ACTION CalculatePowerPerCabinet:

	//If the Cabinet do not exist, do nothing
	IF NOT gInkBox.Status.Cabinets[iCabinet].xExists THEN
		RETURN;
	END_IF

	rPowerPerCabinet := 0;
	FOR iIndex := 1 TO gInkBox.Parameters.Cabinets[iCabinet].TotalInkSystems DO
		rPowerPerCabinet := rPowerPerCabinet + (gInks[iInkIndex].status.Temp.rDutyCycleTemp/100) * gInks[iInkIndex].parameters.parBar.iPowerTempWatt;
		xaExistingInks[iInkIndex] := TRUE;
		iInkIndex := iInkIndex + 1;
	END_FOR
	gInkBox.Status.Cabinets[iCabinet].rTotalAskedPower := rPowerPerCabinet;

END_ACTION

ACTION AssignPowerPerCabinet:

	//If the Cabinet do not exist, do nothing
	IF NOT gInkBox.Status.Cabinets[iCabinet].xExists THEN
		gInkBox.Status.Cabinets[iCabinet].rPowerReduction := 0;
		RETURN;
	END_IF

	//Calculate the reduction in power per cabinet
	IF gInkBox.Status.Cabinets[iCabinet].rTotalAskedPower = 0 THEN
		rCabinetReductionTempPower := 1.0;
	ELSE
		rMaxTempPower := gInkBox.Parameters.Cabinets[iCabinet].MaxTempPowerPsu / gInkBox.Parameters.Cabinets[iCabinet].TotalInksPerPsu;
		rCabinetReductionTempPower:= rMaxTempPower / gInkBox.Status.Cabinets[iCabinet].rTotalAskedPower ;
		rCabinetReductionTempPower:= MIN(rCabinetReductionTempPower, 1.0);
	END_IF
	gInkBox.Status.Cabinets[iCabinet].rPowerReduction := rCabinetReductionTempPower;

	//Assign reduction to inks in cabinet
	FOR iIndex := 1 TO gInkBox.Parameters.Cabinets[iCabinet].TotalInkSystems DO
		gInks[iInkIndex].parameters.Temp.rReductionTempPower:=rCabinetReductionTempPower;
		iInkIndex := iInkIndex + 1;
	END_FOR

END_ACTION
```

#### printHeadData.st - Printhead data parameters
```iecst
ACTION printHeadData:

	IF dataInksInput.parameters.xDebugMode THEN
		dataInksInParams.parBar := gInksPermanentParBar[iIndex];
		RETURN;
	END_IF

	printHeadData_Nozomi2;

END_ACTION
```

#### printHeadBaseData.st
```iecst
ACTION printHeadBaseData:

	// PID MENISCUS values defined by default
	dataInksInParams.parBar.paramsPidMeniscus.rKp:=1.5;
	dataInksInParams.parBar.paramsPidMeniscus.rTi:=10.0;
	dataInksInParams.parBar.paramsPidMeniscus.rKd:=0.01;
	dataInksInParams.parBar.paramsPidMeniscus.rTd:=100;

	//Initial PID POSITIVE values defined by default
	dataInksInParams.parBar.paramsPidPositive.rKp:=0.8;
	dataInksInParams.parBar.paramsPidPositive.rTi:=12;
	dataInksInParams.parBar.paramsPidPositive.rKd:=0.01;
	dataInksInParams.parBar.paramsPidPositive.rTd:=100;

	//Initial PID TEMPERATURE values defined by default
	dataInksInParams.parBar.paramsPidTemp.rKp:=4.0;
	dataInksInParams.parBar.paramsPidTemp.rTi:=250.0;
	dataInksInParams.parBar.paramsPidTemp.rKd:=40.0;
	dataInksInParams.parBar.paramsPidTemp.rTd:=30.0;

	//Initial PID TEMPERATURE values defined by default
	dataInksInParams.parBar.paramsPidTankTemp.rKp:=0.3;
	dataInksInParams.parBar.paramsPidTankTemp.rTi:=32;
	dataInksInParams.parBar.paramsPidTankTemp.rKd:=0;
	dataInksInParams.parBar.paramsPidTankTemp.rTd:=0;

	// Initial PID MENISCUS IN RESERV MODE values defined by default
	dataInksInParams.parBar.paramsPidMeniscusReservoir.rKp:=2.25;
	dataInksInParams.parBar.paramsPidMeniscusReservoir.rTi:=15;
	dataInksInParams.parBar.paramsPidMeniscusReservoir.rKd:=0.01;
	dataInksInParams.parBar.paramsPidMeniscusReservoir.rTd:=100;

	// Initial PID POSITIVE IN RESERV MODE values defined by default
	dataInksInParams.parBar.paramsPidPositiveReservoir.rKp:=0.35;
	dataInksInParams.parBar.paramsPidPositiveReservoir.rTi:=7;
	dataInksInParams.parBar.paramsPidPositiveReservoir.rKd:=0.01;
	dataInksInParams.parBar.paramsPidPositiveReservoir.rTd:=100;

	//Initial PID accelerator temperature params
	dataInksInParams.Temp.rk1Temp := 0.0;
	dataInksInParams.Temp.rk2Temp := 6.0;
	dataInksInParams.Temp.rk3Temp := 2.0;
	dataInksInParams.Temp.rk4Temp := 4.0;

	// It is used in xReservoirModeActivated
	dataInksInParams.parBar.rHighPumpLimitNeg:=5;
	dataInksInParams.parBar.rHighPumpLimitPos:=5;
	dataInksInParams.parBar.rLowPumpLimitNeg:=0;
	dataInksInParams.parBar.rLowPumpLimitPos:=0;

	dataInksInParams.parBar.rAccelerationFillingPump:=1;
	dataInksInParams.parBar.rSPfillingPumpStarting:=30.0;

	// NOZOMITWO-2541 For advance team testing on Alpha
	IF (gMachine.Pt.MachineModel <> Type_NOZ_2_AQ) THEN
		dataInksInParams.parBar.iStabSole:=500;
		dataInksInParams.parBar.iDesahPid:=800;
		dataInksInParams.parBar.iCloseSole:=0;
	END_IF
	dataInksInParams.parBar.xTypeTankSensorAnalog:=FALSE;
	dataInksInParams.parBar.xTypeTankSensorDigital:=TRUE;
	dataInksInParams.parBar.iPowerTempWatt	:=800; //Total Watts of the heater installed
	dataInksInParams.parBar.rVacuumSensorSpan := 300;
	dataInksInParams.parBar.rVacuumSensorOffset := -150;
	dataInksInParams.parBar.iTimeToActiveDcErrorAlarm := T#10s; //10000; //in ms

	dataInksInParams.xReservoirMode := FALSE;
	dataInksInParams.xEnabledTachoSignals := FALSE;
	dataInksInParams.Priming.xSystemNeedsPriming:=FALSE;

	dataInksInParams.parBar.Default.rTemp := 45;
	dataInksInParams.parBar.Default.rMeniscus := 35;
	dataInksInParams.parBar.Default.rPositive := -10;

	dataInksInParams.parBar.StartUp.rMeniscus := 25; // Value when starting
	//dataInksInParams.parBar.StartUp.rPositive := -10; // Value when starting
	dataInksInParams.parBar.StartUp.iSteps := 5; //Step to final value
	dataInksInParams.parBar.StartUp.iSecondsStable := 20; // Time to change
	dataInksInParams.parBar.StartUp.iSecondsUnstable := 3; // Time to change
	dataInksInParams.parBar.StartUp.rMarginToStable := 2;

END_ACTION

ACTION parBaseMineral_SK1536_L:

	printHeadBaseData;

	// PID MENISCUS values defined by default in P4 because it has been worked in C4,D4 and M4
	dataInksInParams.parBar.paramsPidMeniscus.rKp:=2.25;
	dataInksInParams.parBar.paramsPidMeniscus.rTi:=15;
	dataInksInParams.parBar.paramsPidMeniscus.rKd:=0.01;
	dataInksInParams.parBar.paramsPidMeniscus.rTd:=100;

	//Initial PID POSITIVE values defined by default in P4 because it has been worked in C4,D4 and M4
	dataInksInParams.parBar.paramsPidPositive.rKp:=0.4;
	dataInksInParams.parBar.paramsPidPositive.rTi:=7;
	dataInksInParams.parBar.paramsPidPositive.rKd:=0.01;
	dataInksInParams.parBar.paramsPidPositive.rTd:=100;

	//Initial PID TEMPERATURE values defined by default in SHIELD
	dataInksInParams.parBar.paramsPidTemp.rKp:=3.2;
	dataInksInParams.parBar.paramsPidTemp.rTi:=280.0;
	dataInksInParams.parBar.paramsPidTemp.rKd:=45.0;
	dataInksInParams.parBar.paramsPidTemp.rTd:=30.0;

	//Initial PID accelerator temperature params SHIELD
	dataInksInParams.Temp.rk1Temp := 0.0;
	dataInksInParams.Temp.rk2Temp := 4.5;
	dataInksInParams.Temp.rk3Temp := 2.0;
	dataInksInParams.Temp.rk4Temp := 5.0;

	dataInksInParams.xReservoirMode := TRUE;

END_ACTION

ACTION parBaseMineral_Xaar:

	printHeadBaseData;

	//Initial PID TEMPERATURE values defined by default in P4
	dataInksInParams.parBar.paramsPidTemp.rKp:=1.5; // 4.0;
	dataInksInParams.parBar.paramsPidTemp.rTi:=50; //250.0;
	dataInksInParams.parBar.paramsPidTemp.rKd:=40.0;
	dataInksInParams.parBar.paramsPidTemp.rTd:=30.0;

	dataInksInParams.Priming.xSystemNeedsPriming :=TRUE;
	dataInksInParams.PosPump.rSetPointPrimingStarting	:=10;
	dataInksInParams.NegPump.rSetPointPrimingStarting	:=30;
	dataInksInParams.Priming.rThresholdPressure			:=2;
	dataInksInParams.PosPump.rDCThresholdPriming 		:=30.0;

END_ACTION
```

#### printHeadNozomi2.st - Printhead data parameters Nozomi2
```iecst
ACTION printHeadData_Nozomi2:

	CASE dataInksInput.parSw.Config.iInkType OF
		lc_iInkMineral,
		lc_iInkUV:
			printHeadDataNozomi2_Mineral;

		lc_iInkWater:
			printHeadDataNozomi2_Water;

		lc_iInkSolubleSalts:
			dataInksInput.status.iInkState := INKS_STOPPED;

		ELSE
			dataInksInput.status.iInkState := INKS_STOPPED;

	END_CASE

END_ACTION
```

#### printHeadNozomi2Mineral.st - Printhead data parameters Nozomi2 Mineral
```iecst
ACTION printHeadDataNozomi2_Mineral:

	CASE dataInksInput.parSw.Config.iPrintHeadType OF

		lc_iPrintHeadSK1536,
		lc_iPrintHeadSK1536W,
		lc_iPrintHeadTtec,
		lc_iPrintHeadTtecXL,
		lc_iPrintHeadDimatics:
			parNozomi2base;

		lc_iPrintHeadSK1536L,
		lc_iPrintHeadSK1536LW:
			parNozomi2Mineral_SK1536L;

		lc_iPrintHeadX1003,
		lc_iPrintHeadX1003gs40,
		lc_iPrintHeadX2001,
		lc_iPrintHeadX2001gs40:
			parNozomi2Mineral_Xaar;

		lc_iPrintHeadRicoh:
			parNozomi2Uv_Ricoh;

		ELSE
			dataInksInput.status.iInkState := INKS_STOPPED;

	END_CASE

END_ACTION

ACTION baseModificationNozomi2:

	dataInksInParams.parBar.xTypeTankSensorAnalog:=TRUE;
	dataInksInParams.parBar.xTypeTankSensorDigital:=FALSE;

END_ACTION

ACTION parNozomi2base:

	printHeadBaseData;

	baseModificationNozomi2;

END_ACTION

ACTION parNozomi2Mineral_SK1536L:

	parBaseMineral_SK1536_L;

	baseModificationNozomi2;

END_ACTION

ACTION parNozomi2Mineral_Xaar:

	parBaseMineral_Xaar;

	baseModificationNozomi2;

END_ACTION

ACTION parNozomi2Uv_Ricoh:

	parNozomi2base;

	dataInksInParams.parBar.paramsPidMeniscus.rKp:= 0.4;
	dataInksInParams.parBar.paramsPidPositive.rKp:=0.2;

	dataInksInParams.parBar.rVacuumSensorSpan := 1000;
	dataInksInParams.parBar.rVacuumSensorOffset := -500;

	dataInksInParams.parBar.iTimeToActiveDcErrorAlarm := T#60s; //60000; //in ms

END_ACTION
```

### Package Logical/InkBox/PhysicalMapping - Physical inputs assignation

### Program Logical/InkBox/PhysicalMapping/PhysicalMapInputs

#### MappingInputs.st
```iecst
PROGRAM _CYCLIC

	//If in simulation, do not assign physical mapping
	IF gMachine.Pt.ConfigNameID = GC_CONFIG_INKBOX_SIM_ID THEN
		RETURN;
	END_IF

	InputsInkBox;

END_PROGRAM
```

### Program Logical/InkBox/PhysicalMapping/PhysicalMapOutputs (IEC)

#### OutputsInkBox.st - PhysicalOutputs
```iecst
ACTION OutputsInkBox:

	// GROUP _10x
	//X20DOF322_104.DOutput[1] := gInks[1].signals.out.xOutBarResistance;
	X20DOF322_104.DOutput[3] := gInks[1].signals.out.xOutBarResistance;
	X20DOF322_104.DOutput[5] := gInks[1].signals.out.xOutPowPrintHead;
	X20DOF322_104.DOutput[7] := gInks[1].signals.out.xReliefValve;

	//X20DOF322_104.DOutput[2] := gInks[2].signals.out.xOutBarResistance;
	X20DOF322_104.DOutput[4] := gInks[2].signals.out.xOutBarResistance;
	X20DOF322_104.DOutput[6] := gInks[2].signals.out.xOutPowPrintHead;
	X20DOF322_104.DOutput[8] := gInks[2].signals.out.xReliefValve;

	X20AO4622_105.AOutput[1] := gInks[1].signals.out.iDutyCycleNegative;
	X20AO4622_105.AOutput[3] := gInks[1].signals.out.iDutyCycleFilling;

	X20AO4622_105.AOutput[2] := gInks[2].signals.out.iDutyCycleNegative;
	X20AO4622_105.AOutput[4] := gInks[2].signals.out.iDutyCycleFilling;

	// GROUP _20x
	//X20DOF322_204.DOutput[1] := gInks[3].signals.out.xOutBarResistance;
	X20DOF322_204.DOutput[3] := gInks[3].signals.out.xOutBarResistance;
	X20DOF322_204.DOutput[5] := gInks[3].signals.out.xOutPowPrintHead;
	X20DOF322_204.DOutput[7] := gInks[3].signals.out.xReliefValve;

	//X20DOF322_204.DOutput[2] := gInks[4].signals.out.xOutBarResistance;
	X20DOF322_204.DOutput[4] := gInks[4].signals.out.xOutBarResistance;
	X20DOF322_204.DOutput[6] := gInks[4].signals.out.xOutPowPrintHead;
	X20DOF322_204.DOutput[8] := gInks[4].signals.out.xReliefValve;

	X20AO4622_205.AOutput[1] := gInks[3].signals.out.iDutyCycleNegative;
	X20AO4622_205.AOutput[3] := gInks[3].signals.out.iDutyCycleFilling;

	X20AO4622_205.AOutput[2] := gInks[4].signals.out.iDutyCycleNegative;
	X20AO4622_205.AOutput[4] := gInks[4].signals.out.iDutyCycleFilling;

	// GROUP _30x
	//X20DOF322_304.DOutput[1] := gInks[5].signals.out.xOutBarResistance;
	X20DOF322_304.DOutput[3] := gInks[5].signals.out.xOutBarResistance;
	X20DOF322_304.DOutput[5] := gInks[5].signals.out.xOutPowPrintHead;
	X20DOF322_304.DOutput[7] := gInks[5].signals.out.xReliefValve;

	//X20DOF322_304.DOutput[2] := gInks[6].signals.out.xOutBarResistance;
	X20DOF322_304.DOutput[4] := gInks[6].signals.out.xOutBarResistance;
	X20DOF322_304.DOutput[6] := gInks[6].signals.out.xOutPowPrintHead;
	X20DOF322_304.DOutput[8] := gInks[6].signals.out.xReliefValve;

	X20AO4622_305.AOutput[1] := gInks[5].signals.out.iDutyCycleNegative;
	X20AO4622_305.AOutput[3] := gInks[5].signals.out.iDutyCycleFilling;

	X20AO4622_305.AOutput[2] := gInks[6].signals.out.iDutyCycleNegative;
	X20AO4622_305.AOutput[4] := gInks[6].signals.out.iDutyCycleFilling;

END_ACTION
```

### Program Logical/InkBox/HMI/HMI (IEC)

#### Alarms.st
```iecst
ACTION Alarms:

	IF EDGEPOS(gInks[1].Al.xAlrTankDigitalSensorsError) THEN
		MpAlarmXSet(gAlrCore, 'Inks.Alarm.DigSensError_B01');
	ELSIF EDGENEG(gInks[1].Al.xAlrTankDigitalSensorsError) THEN
		MpAlarmXReset(gAlrCore, 'Inks.Alarm.DigSensError_B01');
	END_IF

	IF EDGEPOS(gInks[1].Al.xAlrVacuum1) THEN
		MpAlarmXSet(gAlrCore, 'Inks.Alarm.xAlrVacuum1_B01');
	ELSIF EDGENEG(gInks[1].Al.xAlrVacuum1) THEN
		MpAlarmXReset(gAlrCore, 'Inks.Alarm.xAlrVacuum1_B01');
	END_IF

	IF EDGEPOS(gInks[1].Al.xAlrVacuum2) THEN
		MpAlarmXSet(gAlrCore, 'Inks.Alarm.xAlrVacuum2_B01');
	ELSIF EDGENEG(gInks[1].Al.xAlrVacuum2) THEN
		MpAlarmXReset(gAlrCore, 'Inks.Alarm.xAlrVacuum2_B01');
	END_IF

	IF EDGEPOS(gInks[1].Al.xAlrVacuumSensor1) THEN
		MpAlarmXSet(gAlrCore, 'Inks.Alarm.inks.Al.xAlrVacuumSensor1_B01');
	ELSIF EDGENEG(gInks[1].Al.xAlrVacuumSensor1) THEN
		MpAlarmXReset(gAlrCore, 'Inks.Alarm.inks.Al.xAlrVacuumSensor1_B01');
	END_IF

	IF EDGEPOS(gInks[1].Al.xAlrVacuumSensor2) THEN
		MpAlarmXSet(gAlrCore, 'Inks.Alarm.inks.Al.xAlrVacuumSensor2_B01');
	ELSIF EDGENEG(gInks[1].Al.xAlrVacuumSensor2) THEN
		MpAlarmXReset(gAlrCore, 'Inks.Alarm.inks.Al.xAlrVacuumSensor2_B01');
	END_IF

	IF EDGEPOS(gInks[1].Al.xAlrDiffVacuum) THEN
		MpAlarmXSet(gAlrCore, 'Inks.Alarm.inks.Al.xAlrDiffVacuum_B01');
	ELSIF EDGENEG(gInks[1].Al.xAlrDiffVacuum) THEN
		MpAlarmXReset(gAlrCore, 'Inks.Alarm.inks.Al.xAlrDiffVacuum_B01');
	END_IF

	IF EDGEPOS(gInks[1].Al.xAlrIncoherTempHeat) THEN
		MpAlarmXSet(gAlrCore, 'Inks.Alarm.inks.Al.xAlrIncoherTempHeat_B01');
	ELSIF EDGENEG(gInks[1].Al.xAlrIncoherTempHeat) THEN
		MpAlarmXReset(gAlrCore, 'Inks.Alarm.inks.Al.xAlrIncoherTempHeat_B01');
	END_IF

	IF EDGEPOS(gInks[1].Al.xAlrHeaterReachsMaxTemp) THEN
		MpAlarmXSet(gAlrCore, 'Inks.Alarm.inks.Al.xAlrHeaterReachsMaxTemp_B01');
	ELSIF EDGENEG(gInks[1].Al.xAlrHeaterReachsMaxTemp) THEN
		MpAlarmXReset(gAlrCore, 'Inks.Alarm.inks.Al.xAlrHeaterReachsMaxTemp_B01');
	END_IF

	IF EDGEPOS(gInks[1].Al.xAlrTempSensor) THEN
		MpAlarmXSet(gAlrCore, 'Inks.Alarm.inks.Al.xAlrTempSensor_B01');
	ELSIF EDGENEG(gInks[1].Al.xAlrTempSensor) THEN
		MpAlarmXReset(gAlrCore, 'Inks.Alarm.inks.Al.xAlrTempSensor_B01');
	END_IF

	IF EDGEPOS(gInks[1].Al.xAlrDiffInCtrlTemp) THEN
		MpAlarmXSet(gAlrCore, 'Inks.Alarm.inks.Al.xAlrDiffInCtrlTemp_B01');
	ELSIF EDGENEG(gInks[1].Al.xAlrDiffInCtrlTemp) THEN
		MpAlarmXReset(gAlrCore, 'Inks.Alarm.inks.Al.xAlrDiffInCtrlTemp_B01');
	END_IF

	IF EDGEPOS(gInks[1].Al.xAlrDifCtrlTempExcessive) THEN
		MpAlarmXSet(gAlrCore, 'Inks.Alarm.inks.Al.xAlrDifCtrlTempExcessive_B01');
	ELSIF EDGENEG(gInks[1].Al.xAlrDifCtrlTempExcessive) THEN
		MpAlarmXReset(gAlrCore, 'Inks.Alarm.inks.Al.xAlrDifCtrlTempExcessive_B01');
	END_IF

	IF EDGEPOS(gInks[1].Al.xAlrHeaterOutFault) THEN
		MpAlarmXSet(gAlrCore, 'Inks.Alarm.inks.Al.xAlrHeaterOutFault_B01');
	ELSIF EDGENEG(gInks[1].Al.xAlrHeaterOutFault) THEN
		MpAlarmXReset(gAlrCore, 'Inks.Alarm.inks.Al.xAlrHeaterOutFault_B01');
	END_IF

	IF EDGEPOS(gInks[1].Al.xAlrOverPressure) THEN
		MpAlarmXSet(gAlrCore, 'Inks.Alarm.inks.Al.xAlrOverPressure_B01');
	ELSIF EDGENEG(gInks[1].Al.xAlrOverPressure) THEN
		MpAlarmXReset(gAlrCore, 'Inks.Alarm.inks.Al.xAlrOverPressure_B01');
	END_IF

	IF EDGEPOS(gInks[1].Al.xAlrStopRecircNoInk) THEN
		MpAlarmXSet(gAlrCore, 'Inks.Alarm.inks.Al.xAlrStopRecircNoInk_B01');
	ELSIF EDGENEG(gInks[1].Al.xAlrStopRecircNoInk) THEN
		MpAlarmXReset(gAlrCore, 'Inks.Alarm.inks.Al.xAlrStopRecircNoInk_B01');
	END_IF

	IF EDGEPOS(gInks[1].Al.xAlrBrokenMeniscus) THEN
		MpAlarmXSet(gAlrCore, 'Inks.Alarm.inks.Al.xAlrBrokenMeniscus_B01');
	ELSIF EDGENEG(gInks[1].Al.xAlrBrokenMeniscus) THEN
		MpAlarmXReset(gAlrCore, 'Inks.Alarm.inks.Al.xAlrBrokenMeniscus_B01');
	END_IF

	IF EDGEPOS(gInks[1].Al.xAlrLevelSensorError) THEN
		MpAlarmXSet(gAlrCore, 'Inks.Alarm.inks.Al.xAlrLevelSensorError_B01');
	ELSIF EDGENEG(gInks[1].Al.xAlrLevelSensorError) THEN
		MpAlarmXReset(gAlrCore, 'Inks.Alarm.inks.Al.xAlrLevelSensorError_B01');
	END_IF

	IF EDGEPOS(gInks[1].Al.xAlrTankEmpty) THEN
		MpAlarmXSet(gAlrCore, 'Inks.Alarm.inks.Al.xAlrTankEmpty_B01');
	ELSIF EDGENEG(gInks[1].Al.xAlrTankEmpty) THEN
		MpAlarmXReset(gAlrCore, 'Inks.Alarm.inks.Al.xAlrTankEmpty_B01');
	END_IF

	IF EDGEPOS(gInks[1].Al.xAlrTankToFillIn) THEN
		MpAlarmXSet(gAlrCore, 'Inks.Alarm.inks.Al.xAlrTankToFillIn_B01');
	ELSIF EDGENEG(gInks[1].Al.xAlrTankToFillIn) THEN
		MpAlarmXReset(gAlrCore, 'Inks.Alarm.inks.Al.xAlrTankToFillIn_B01');
	END_IF

	IF EDGEPOS(gInks[1].Al.xAlrPumpsDCError) THEN
		MpAlarmXSet(gAlrCore, 'Inks.Alarm.inks.Al.xAlrPumpsDCError_B01');
	ELSIF EDGENEG(gInks[1].Al.xAlrPumpsDCError) THEN
		MpAlarmXReset(gAlrCore, 'Inks.Alarm.inks.Al.xAlrPumpsDCError_B01');
	END_IF

	IF EDGEPOS(gInks[1].Al.xAlrKlixonTriggered) THEN
		MpAlarmXSet(gAlrCore, 'Inks.Alarm.inks.Al.xAlrKlixonTriggered_B01');
	ELSIF EDGENEG(gInks[1].Al.xAlrKlixonTriggered) THEN
		MpAlarmXReset(gAlrCore, 'Inks.Alarm.inks.Al.xAlrKlixonTriggered_B01');
	END_IF

	IF EDGEPOS(gInks[1].Al.xAlrPrintHeadPsuFailure) THEN
		MpAlarmXSet(gAlrCore, 'Inks.Alarm.inks.Al.xAlrPrintHeadPsuFailure_B01');
	ELSIF EDGENEG(gInks[1].Al.xAlrPrintHeadPsuFailure) THEN
		MpAlarmXReset(gAlrCore, 'Inks.Alarm.inks.Al.xAlrPrintHeadPsuFailure_B01');
	END_IF

	IF EDGEPOS(gInks[2].Al.xAlrTankDigitalSensorsError) THEN
		MpAlarmXSet(gAlrCore, 'Inks.Alarm.DigSensError_B02');
	ELSIF EDGENEG(gInks[2].Al.xAlrTankDigitalSensorsError) THEN
		MpAlarmXReset(gAlrCore, 'Inks.Alarm.DigSensError_B02');
	END_IF

	IF EDGEPOS(gInks[2].Al.xAlrVacuum1) THEN
		MpAlarmXSet(gAlrCore, 'Inks.Alarm.xAlrVacuum1_B02');
	ELSIF EDGENEG(gInks[2].Al.xAlrVacuum1) THEN
		MpAlarmXReset(gAlrCore, 'Inks.Alarm.xAlrVacuum1_B02');
	END_IF

	IF EDGEPOS(gInks[2].Al.xAlrVacuum2) THEN
		MpAlarmXSet(gAlrCore, 'Inks.Alarm.xAlrVacuum2_B02');
	ELSIF EDGENEG(gInks[2].Al.xAlrVacuum2) THEN
		MpAlarmXReset(gAlrCore, 'Inks.Alarm.xAlrVacuum2_B02');
	END_IF

	IF EDGEPOS(gInks[2].Al.xAlrVacuumSensor1) THEN
		MpAlarmXSet(gAlrCore, 'Inks.Alarm.inks.Al.xAlrVacuumSensor1_B02');
	ELSIF EDGENEG(gInks[2].Al.xAlrVacuumSensor1) THEN
		MpAlarmXReset(gAlrCore, 'Inks.Alarm.inks.Al.xAlrVacuumSensor1_B02');
	END_IF

	IF EDGEPOS(gInks[2].Al.xAlrVacuumSensor2) THEN
		MpAlarmXSet(gAlrCore, 'Inks.Alarm.inks.Al.xAlrVacuumSensor2_B02');
	ELSIF EDGENEG(gInks[2].Al.xAlrVacuumSensor2) THEN
		MpAlarmXReset(gAlrCore, 'Inks.Alarm.inks.Al.xAlrVacuumSensor2_B02');
	END_IF

	IF EDGEPOS(gInks[2].Al.xAlrDiffVacuum) THEN
		MpAlarmXSet(gAlrCore, 'Inks.Alarm.inks.Al.xAlrDiffVacuum_B02');
	ELSIF EDGENEG(gInks[2].Al.xAlrDiffVacuum) THEN
		MpAlarmXReset(gAlrCore, 'Inks.Alarm.inks.Al.xAlrDiffVacuum_B02');
	END_IF

	IF EDGEPOS(gInks[2].Al.xAlrIncoherTempHeat) THEN
		MpAlarmXSet(gAlrCore, 'Inks.Alarm.inks.Al.xAlrIncoherTempHeat_B02');
	ELSIF EDGENEG(gInks[2].Al.xAlrIncoherTempHeat) THEN
		MpAlarmXReset(gAlrCore, 'Inks.Alarm.inks.Al.xAlrIncoherTempHeat_B02');
	END_IF

	IF EDGEPOS(gInks[2].Al.xAlrHeaterReachsMaxTemp) THEN
		MpAlarmXSet(gAlrCore, 'Inks.Alarm.inks.Al.xAlrHeaterReachsMaxTemp_B02');
	ELSIF EDGENEG(gInks[2].Al.xAlrHeaterReachsMaxTemp) THEN
		MpAlarmXReset(gAlrCore, 'Inks.Alarm.inks.Al.xAlrHeaterReachsMaxTemp_B02');
	END_IF

	IF EDGEPOS(gInks[2].Al.xAlrTempSensor) THEN
		MpAlarmXSet(gAlrCore, 'Inks.Alarm.inks.Al.xAlrTempSensor_B02');
	ELSIF EDGENEG(gInks[2].Al.xAlrTempSensor) THEN
		MpAlarmXReset(gAlrCore, 'Inks.Alarm.inks.Al.xAlrTempSensor_B02');
	END_IF

	IF EDGEPOS(gInks[2].Al.xAlrDiffInCtrlTemp) THEN
		MpAlarmXSet(gAlrCore, 'Inks.Alarm.inks.Al.xAlrDiffInCtrlTemp_B02');
	ELSIF EDGENEG(gInks[2].Al.xAlrDiffInCtrlTemp) THEN
		MpAlarmXReset(gAlrCore, 'Inks.Alarm.inks.Al.xAlrDiffInCtrlTemp_B02');
	END_IF

	IF EDGEPOS(gInks[2].Al.xAlrDifCtrlTempExcessive) THEN
		MpAlarmXSet(gAlrCore, 'Inks.Alarm.inks.Al.xAlrDifCtrlTempExcessive_B02');
	ELSIF EDGENEG(gInks[2].Al.xAlrDifCtrlTempExcessive) THEN
		MpAlarmXReset(gAlrCore, 'Inks.Alarm.inks.Al.xAlrDifCtrlTempExcessive_B02');
	END_IF

	IF EDGEPOS(gInks[2].Al.xAlrHeaterOutFault) THEN
		MpAlarmXSet(gAlrCore, 'Inks.Alarm.inks.Al.xAlrHeaterOutFault_B02');
	ELSIF EDGENEG(gInks[2].Al.xAlrHeaterOutFault) THEN
		MpAlarmXReset(gAlrCore, 'Inks.Alarm.inks.Al.xAlrHeaterOutFault_B02');
	END_IF

	IF EDGEPOS(gInks[2].Al.xAlrOverPressure) THEN
		MpAlarmXSet(gAlrCore, 'Inks.Alarm.inks.Al.xAlrOverPressure_B02');
	ELSIF EDGENEG(gInks[2].Al.xAlrOverPressure) THEN
		MpAlarmXReset(gAlrCore, 'Inks.Alarm.inks.Al.xAlrOverPressure_B02');
	END_IF

	IF EDGEPOS(gInks[2].Al.xAlrStopRecircNoInk) THEN
		MpAlarmXSet(gAlrCore, 'Inks.Alarm.inks.Al.xAlrStopRecircNoInk_B02');
	ELSIF EDGENEG(gInks[2].Al.xAlrStopRecircNoInk) THEN
		MpAlarmXReset(gAlrCore, 'Inks.Alarm.inks.Al.xAlrStopRecircNoInk_B02');
	END_IF

	IF EDGEPOS(gInks[2].Al.xAlrBrokenMeniscus) THEN
		MpAlarmXSet(gAlrCore, 'Inks.Alarm.inks.Al.xAlrBrokenMeniscus_B02');
	ELSIF EDGENEG(gInks[2].Al.xAlrBrokenMeniscus) THEN
		MpAlarmXReset(gAlrCore, 'Inks.Alarm.inks.Al.xAlrBrokenMeniscus_B02');
	END_IF

	IF EDGEPOS(gInks[2].Al.xAlrLevelSensorError) THEN
		MpAlarmXSet(gAlrCore, 'Inks.Alarm.inks.Al.xAlrLevelSensorError_B02');
	ELSIF EDGENEG(gInks[2].Al.xAlrLevelSensorError) THEN
		MpAlarmXReset(gAlrCore, 'Inks.Alarm.inks.Al.xAlrLevelSensorError_B02');
	END_IF

	IF EDGEPOS(gInks[2].Al.xAlrTankEmpty) THEN
		MpAlarmXSet(gAlrCore, 'Inks.Alarm.inks.Al.xAlrTankEmpty_B02');
	ELSIF EDGENEG(gInks[2].Al.xAlrTankEmpty) THEN
		MpAlarmXReset(gAlrCore, 'Inks.Alarm.inks.Al.xAlrTankEmpty_B02');
	END_IF

	IF EDGEPOS(gInks[2].Al.xAlrTankToFillIn) THEN
		MpAlarmXSet(gAlrCore, 'Inks.Alarm.inks.Al.xAlrTankToFillIn_B02');
	ELSIF EDGENEG(gInks[2].Al.xAlrTankToFillIn) THEN
		MpAlarmXReset(gAlrCore, 'Inks.Alarm.inks.Al.xAlrTankToFillIn_B02');
	END_IF

	IF EDGEPOS(gInks[2].Al.xAlrPumpsDCError) THEN
		MpAlarmXSet(gAlrCore, 'Inks.Alarm.inks.Al.xAlrPumpsDCError_B02');
	ELSIF EDGENEG(gInks[2].Al.xAlrPumpsDCError) THEN
		MpAlarmXReset(gAlrCore, 'Inks.Alarm.inks.Al.xAlrPumpsDCError_B02');
	END_IF

	IF EDGEPOS(gInks[2].Al.xAlrKlixonTriggered) THEN
		MpAlarmXSet(gAlrCore, 'Inks.Alarm.inks.Al.xAlrKlixonTriggered_B02');
	ELSIF EDGENEG(gInks[2].Al.xAlrKlixonTriggered) THEN
		MpAlarmXReset(gAlrCore, 'Inks.Alarm.inks.Al.xAlrKlixonTriggered_B02');
	END_IF

	IF EDGEPOS(gInks[2].Al.xAlrPrintHeadPsuFailure) THEN
		MpAlarmXSet(gAlrCore, 'Inks.Alarm.inks.Al.xAlrPrintHeadPsuFailure_B02');
	ELSIF EDGENEG(gInks[2].Al.xAlrPrintHeadPsuFailure) THEN
		MpAlarmXReset(gAlrCore, 'Inks.Alarm.inks.Al.xAlrPrintHeadPsuFailure_B02');
	END_IF

	IF EDGEPOS(gInks[3].Al.xAlrTankDigitalSensorsError) THEN
		MpAlarmXSet(gAlrCore, 'Inks.Alarm.DigSensError_B03');
	ELSIF EDGENEG(gInks[3].Al.xAlrTankDigitalSensorsError) THEN
		MpAlarmXReset(gAlrCore, 'Inks.Alarm.DigSensError_B03');
	END_IF

	IF EDGEPOS(gInks[3].Al.xAlrVacuum1) THEN
		MpAlarmXSet(gAlrCore, 'Inks.Alarm.xAlrVacuum1_B03');
	ELSIF EDGENEG(gInks[3].Al.xAlrVacuum1) THEN
		MpAlarmXReset(gAlrCore, 'Inks.Alarm.xAlrVacuum1_B03');
	END_IF

	IF EDGEPOS(gInks[3].Al.xAlrVacuum2) THEN
		MpAlarmXSet(gAlrCore, 'Inks.Alarm.xAlrVacuum2_B03');
	ELSIF EDGENEG(gInks[3].Al.xAlrVacuum2) THEN
		MpAlarmXReset(gAlrCore, 'Inks.Alarm.xAlrVacuum2_B03');
	END_IF

	IF EDGEPOS(gInks[3].Al.xAlrVacuumSensor1) THEN
		MpAlarmXSet(gAlrCore, 'Inks.Alarm.inks.Al.xAlrVacuumSensor1_B03');
	ELSIF EDGENEG(gInks[3].Al.xAlrVacuumSensor1) THEN
		MpAlarmXReset(gAlrCore, 'Inks.Alarm.inks.Al.xAlrVacuumSensor1_B03');
	END_IF

	IF EDGEPOS(gInks[3].Al.xAlrVacuumSensor2) THEN
		MpAlarmXSet(gAlrCore, 'Inks.Alarm.inks.Al.xAlrVacuumSensor2_B03');
	ELSIF EDGENEG(gInks[3].Al.xAlrVacuumSensor2) THEN
		MpAlarmXReset(gAlrCore, 'Inks.Alarm.inks.Al.xAlrVacuumSensor2_B03');
	END_IF

	IF EDGEPOS(gInks[3].Al.xAlrDiffVacuum) THEN
		MpAlarmXSet(gAlrCore, 'Inks.Alarm.inks.Al.xAlrDiffVacuum_B03');
	ELSIF EDGENEG(gInks[3].Al.xAlrDiffVacuum) THEN
		MpAlarmXReset(gAlrCore, 'Inks.Alarm.inks.Al.xAlrDiffVacuum_B03');
	END_IF

	IF EDGEPOS(gInks[3].Al.xAlrIncoherTempHeat) THEN
		MpAlarmXSet(gAlrCore, 'Inks.Alarm.inks.Al.xAlrIncoherTempHeat_B03');
	ELSIF EDGENEG(gInks[3].Al.xAlrIncoherTempHeat) THEN
		MpAlarmXReset(gAlrCore, 'Inks.Alarm.inks.Al.xAlrIncoherTempHeat_B03');
	END_IF

	IF EDGEPOS(gInks[3].Al.xAlrHeaterReachsMaxTemp) THEN
		MpAlarmXSet(gAlrCore, 'Inks.Alarm.inks.Al.xAlrHeaterReachsMaxTemp_B03');
	ELSIF EDGENEG(gInks[3].Al.xAlrHeaterReachsMaxTemp) THEN
		MpAlarmXReset(gAlrCore, 'Inks.Alarm.inks.Al.xAlrHeaterReachsMaxTemp_B03');
	END_IF

	IF EDGEPOS(gInks[3].Al.xAlrTempSensor) THEN
		MpAlarmXSet(gAlrCore, 'Inks.Alarm.inks.Al.xAlrTempSensor_B03');
	ELSIF EDGENEG(gInks[3].Al.xAlrTempSensor) THEN
		MpAlarmXReset(gAlrCore, 'Inks.Alarm.inks.Al.xAlrTempSensor_B03');
	END_IF

	IF EDGEPOS(gInks[3].Al.xAlrDiffInCtrlTemp) THEN
		MpAlarmXSet(gAlrCore, 'Inks.Alarm.inks.Al.xAlrDiffInCtrlTemp_B03');
	ELSIF EDGENEG(gInks[3].Al.xAlrDiffInCtrlTemp) THEN
		MpAlarmXReset(gAlrCore, 'Inks.Alarm.inks.Al.xAlrDiffInCtrlTemp_B03');
	END_IF

	IF EDGEPOS(gInks[3].Al.xAlrDifCtrlTempExcessive) THEN
		MpAlarmXSet(gAlrCore, 'Inks.Alarm.inks.Al.xAlrDifCtrlTempExcessive_B03');
	ELSIF EDGENEG(gInks[3].Al.xAlrDifCtrlTempExcessive) THEN
		MpAlarmXReset(gAlrCore, 'Inks.Alarm.inks.Al.xAlrDifCtrlTempExcessive_B03');
	END_IF

	IF EDGEPOS(gInks[3].Al.xAlrHeaterOutFault) THEN
		MpAlarmXSet(gAlrCore, 'Inks.Alarm.inks.Al.xAlrHeaterOutFault_B03');
	ELSIF EDGENEG(gInks[3].Al.xAlrHeaterOutFault) THEN
		MpAlarmXReset(gAlrCore, 'Inks.Alarm.inks.Al.xAlrHeaterOutFault_B03');
	END_IF

	IF EDGEPOS(gInks[3].Al.xAlrOverPressure) THEN
		MpAlarmXSet(gAlrCore, 'Inks.Alarm.inks.Al.xAlrOverPressure_B03');
	ELSIF EDGENEG(gInks[3].Al.xAlrOverPressure) THEN
		MpAlarmXReset(gAlrCore, 'Inks.Alarm.inks.Al.xAlrOverPressure_B03');
	END_IF

	IF EDGEPOS(gInks[3].Al.xAlrStopRecircNoInk) THEN
		MpAlarmXSet(gAlrCore, 'Inks.Alarm.inks.Al.xAlrStopRecircNoInk_B03');
	ELSIF EDGENEG(gInks[3].Al.xAlrStopRecircNoInk) THEN
		MpAlarmXReset(gAlrCore, 'Inks.Alarm.inks.Al.xAlrStopRecircNoInk_B03');
	END_IF

	IF EDGEPOS(gInks[3].Al.xAlrBrokenMeniscus) THEN
		MpAlarmXSet(gAlrCore, 'Inks.Alarm.inks.Al.xAlrBrokenMeniscus_B03');
	ELSIF EDGENEG(gInks[3].Al.xAlrBrokenMeniscus) THEN
		MpAlarmXReset(gAlrCore, 'Inks.Alarm.inks.Al.xAlrBrokenMeniscus_B03');
	END_IF

	IF EDGEPOS(gInks[3].Al.xAlrLevelSensorError) THEN
		MpAlarmXSet(gAlrCore, 'Inks.Alarm.inks.Al.xAlrLevelSensorError_B03');
	ELSIF EDGENEG(gInks[3].Al.xAlrLevelSensorError) THEN
		MpAlarmXReset(gAlrCore, 'Inks.Alarm.inks.Al.xAlrLevelSensorError_B03');
	END_IF

	IF EDGEPOS(gInks[3].Al.xAlrTankEmpty) THEN
		MpAlarmXSet(gAlrCore, 'Inks.Alarm.inks.Al.xAlrTankEmpty_B03');
	ELSIF EDGENEG(gInks[3].Al.xAlrTankEmpty) THEN
		MpAlarmXReset(gAlrCore, 'Inks.Alarm.inks.Al.xAlrTankEmpty_B03');
	END_IF

	IF EDGEPOS(gInks[3].Al.xAlrTankToFillIn) THEN
		MpAlarmXSet(gAlrCore, 'Inks.Alarm.inks.Al.xAlrTankToFillIn_B03');
	ELSIF EDGENEG(gInks[3].Al.xAlrTankToFillIn) THEN
		MpAlarmXReset(gAlrCore, 'Inks.Alarm.inks.Al.xAlrTankToFillIn_B03');
	END_IF

	IF EDGEPOS(gInks[3].Al.xAlrPumpsDCError) THEN
		MpAlarmXSet(gAlrCore, 'Inks.Alarm.inks.Al.xAlrPumpsDCError_B03');
	ELSIF EDGENEG(gInks[3].Al.xAlrPumpsDCError) THEN
		MpAlarmXReset(gAlrCore, 'Inks.Alarm.inks.Al.xAlrPumpsDCError_B03');
	END_IF

	IF EDGEPOS(gInks[3].Al.xAlrKlixonTriggered) THEN
		MpAlarmXSet(gAlrCore, 'Inks.Alarm.inks.Al.xAlrKlixonTriggered_B03');
	ELSIF EDGENEG(gInks[3].Al.xAlrKlixonTriggered) THEN
		MpAlarmXReset(gAlrCore, 'Inks.Alarm.inks.Al.xAlrKlixonTriggered_B03');
	END_IF

	IF EDGEPOS(gInks[3].Al.xAlrPrintHeadPsuFailure) THEN
		MpAlarmXSet(gAlrCore, 'Inks.Alarm.inks.Al.xAlrPrintHeadPsuFailure_B03');
	ELSIF EDGENEG(gInks[3].Al.xAlrPrintHeadPsuFailure) THEN
		MpAlarmXReset(gAlrCore, 'Inks.Alarm.inks.Al.xAlrPrintHeadPsuFailure_B03');
	END_IF

	IF EDGEPOS(gInks[4].Al.xAlrTankDigitalSensorsError) THEN
		MpAlarmXSet(gAlrCore, 'Inks.Alarm.DigSensError_B04');
	ELSIF EDGENEG(gInks[4].Al.xAlrTankDigitalSensorsError) THEN
		MpAlarmXReset(gAlrCore, 'Inks.Alarm.DigSensError_B04');
	END_IF

	IF EDGEPOS(gInks[4].Al.xAlrVacuum1) THEN
		MpAlarmXSet(gAlrCore, 'Inks.Alarm.xAlrVacuum1_B04');
	ELSIF EDGENEG(gInks[4].Al.xAlrVacuum1) THEN
		MpAlarmXReset(gAlrCore, 'Inks.Alarm.xAlrVacuum1_B04');
	END_IF

	IF EDGEPOS(gInks[4].Al.xAlrVacuum2) THEN
		MpAlarmXSet(gAlrCore, 'Inks.Alarm.xAlrVacuum2_B04');
	ELSIF EDGENEG(gInks[4].Al.xAlrVacuum2) THEN
		MpAlarmXReset(gAlrCore, 'Inks.Alarm.xAlrVacuum2_B04');
	END_IF

	IF EDGEPOS(gInks[4].Al.xAlrVacuumSensor1) THEN
		MpAlarmXSet(gAlrCore, 'Inks.Alarm.inks.Al.xAlrVacuumSensor1_B04');
	ELSIF EDGENEG(gInks[4].Al.xAlrVacuumSensor1) THEN
		MpAlarmXReset(gAlrCore, 'Inks.Alarm.inks.Al.xAlrVacuumSensor1_B04');
	END_IF

	IF EDGEPOS(gInks[4].Al.xAlrVacuumSensor2) THEN
		MpAlarmXSet(gAlrCore, 'Inks.Alarm.inks.Al.xAlrVacuumSensor2_B04');
	ELSIF EDGENEG(gInks[4].Al.xAlrVacuumSensor2) THEN
		MpAlarmXReset(gAlrCore, 'Inks.Alarm.inks.Al.xAlrVacuumSensor2_B04');
	END_IF

	IF EDGEPOS(gInks[4].Al.xAlrDiffVacuum) THEN
		MpAlarmXSet(gAlrCore, 'Inks.Alarm.inks.Al.xAlrDiffVacuum_B04');
	ELSIF EDGENEG(gInks[4].Al.xAlrDiffVacuum) THEN
		MpAlarmXReset(gAlrCore, 'Inks.Alarm.inks.Al.xAlrDiffVacuum_B04');
	END_IF

	IF EDGEPOS(gInks[4].Al.xAlrIncoherTempHeat) THEN
		MpAlarmXSet(gAlrCore, 'Inks.Alarm.inks.Al.xAlrIncoherTempHeat_B04');
	ELSIF EDGENEG(gInks[4].Al.xAlrIncoherTempHeat) THEN
		MpAlarmXReset(gAlrCore, 'Inks.Alarm.inks.Al.xAlrIncoherTempHeat_B04');
	END_IF

	IF EDGEPOS(gInks[4].Al.xAlrHeaterReachsMaxTemp) THEN
		MpAlarmXSet(gAlrCore, 'Inks.Alarm.inks.Al.xAlrHeaterReachsMaxTemp_B04');
	ELSIF EDGENEG(gInks[4].Al.xAlrHeaterReachsMaxTemp) THEN
		MpAlarmXReset(gAlrCore, 'Inks.Alarm.inks.Al.xAlrHeaterReachsMaxTemp_B04');
	END_IF

	IF EDGEPOS(gInks[4].Al.xAlrTempSensor) THEN
		MpAlarmXSet(gAlrCore, 'Inks.Alarm.inks.Al.xAlrTempSensor_B04');
	ELSIF EDGENEG(gInks[4].Al.xAlrTempSensor) THEN
		MpAlarmXReset(gAlrCore, 'Inks.Alarm.inks.Al.xAlrTempSensor_B04');
	END_IF

	IF EDGEPOS(gInks[4].Al.xAlrDiffInCtrlTemp) THEN
		MpAlarmXSet(gAlrCore, 'Inks.Alarm.inks.Al.xAlrDiffInCtrlTemp_B04');
	ELSIF EDGENEG(gInks[4].Al.xAlrDiffInCtrlTemp) THEN
		MpAlarmXReset(gAlrCore, 'Inks.Alarm.inks.Al.xAlrDiffInCtrlTemp_B04');
	END_IF

	IF EDGEPOS(gInks[4].Al.xAlrDifCtrlTempExcessive) THEN
		MpAlarmXSet(gAlrCore, 'Inks.Alarm.inks.Al.xAlrDifCtrlTempExcessive_B04');
	ELSIF EDGENEG(gInks[4].Al.xAlrDifCtrlTempExcessive) THEN
		MpAlarmXReset(gAlrCore, 'Inks.Alarm.inks.Al.xAlrDifCtrlTempExcessive_B04');
	END_IF

	IF EDGEPOS(gInks[4].Al.xAlrHeaterOutFault) THEN
		MpAlarmXSet(gAlrCore, 'Inks.Alarm.inks.Al.xAlrHeaterOutFault_B04');
	ELSIF EDGENEG(gInks[4].Al.xAlrHeaterOutFault) THEN
		MpAlarmXReset(gAlrCore, 'Inks.Alarm.inks.Al.xAlrHeaterOutFault_B04');
	END_IF

	IF EDGEPOS(gInks[4].Al.xAlrOverPressure) THEN
		MpAlarmXSet(gAlrCore, 'Inks.Alarm.inks.Al.xAlrOverPressure_B04');
	ELSIF EDGENEG(gInks[4].Al.xAlrOverPressure) THEN
		MpAlarmXReset(gAlrCore, 'Inks.Alarm.inks.Al.xAlrOverPressure_B04');
	END_IF

	IF EDGEPOS(gInks[4].Al.xAlrStopRecircNoInk) THEN
		MpAlarmXSet(gAlrCore, 'Inks.Alarm.inks.Al.xAlrStopRecircNoInk_B04');
	ELSIF EDGENEG(gInks[4].Al.xAlrStopRecircNoInk) THEN
		MpAlarmXReset(gAlrCore, 'Inks.Alarm.inks.Al.xAlrStopRecircNoInk_B04');
	END_IF

	IF EDGEPOS(gInks[4].Al.xAlrBrokenMeniscus) THEN
		MpAlarmXSet(gAlrCore, 'Inks.Alarm.inks.Al.xAlrBrokenMeniscus_B04');
	ELSIF EDGENEG(gInks[4].Al.xAlrBrokenMeniscus) THEN
		MpAlarmXReset(gAlrCore, 'Inks.Alarm.inks.Al.xAlrBrokenMeniscus_B04');
	END_IF

	IF EDGEPOS(gInks[4].Al.xAlrLevelSensorError) THEN
		MpAlarmXSet(gAlrCore, 'Inks.Alarm.inks.Al.xAlrLevelSensorError_B04');
	ELSIF EDGENEG(gInks[4].Al.xAlrLevelSensorError) THEN
		MpAlarmXReset(gAlrCore, 'Inks.Alarm.inks.Al.xAlrLevelSensorError_B04');
	END_IF

	IF EDGEPOS(gInks[4].Al.xAlrTankEmpty) THEN
		MpAlarmXSet(gAlrCore, 'Inks.Alarm.inks.Al.xAlrTankEmpty_B04');
	ELSIF EDGENEG(gInks[4].Al.xAlrTankEmpty) THEN
		MpAlarmXReset(gAlrCore, 'Inks.Alarm.inks.Al.xAlrTankEmpty_B04');
	END_IF

	IF EDGEPOS(gInks[4].Al.xAlrTankToFillIn) THEN
		MpAlarmXSet(gAlrCore, 'Inks.Alarm.inks.Al.xAlrTankToFillIn_B04');
	ELSIF EDGENEG(gInks[4].Al.xAlrTankToFillIn) THEN
		MpAlarmXReset(gAlrCore, 'Inks.Alarm.inks.Al.xAlrTankToFillIn_B04');
	END_IF

	IF EDGEPOS(gInks[4].Al.xAlrPumpsDCError) THEN
		MpAlarmXSet(gAlrCore, 'Inks.Alarm.inks.Al.xAlrPumpsDCError_B04');
	ELSIF EDGENEG(gInks[4].Al.xAlrPumpsDCError) THEN
		MpAlarmXReset(gAlrCore, 'Inks.Alarm.inks.Al.xAlrPumpsDCError_B04');
	END_IF

	IF EDGEPOS(gInks[4].Al.xAlrKlixonTriggered) THEN
		MpAlarmXSet(gAlrCore, 'Inks.Alarm.inks.Al.xAlrKlixonTriggered_B04');
	ELSIF EDGENEG(gInks[4].Al.xAlrKlixonTriggered) THEN
		MpAlarmXReset(gAlrCore, 'Inks.Alarm.inks.Al.xAlrKlixonTriggered_B04');
	END_IF

	IF EDGEPOS(gInks[4].Al.xAlrPrintHeadPsuFailure) THEN
		MpAlarmXSet(gAlrCore, 'Inks.Alarm.inks.Al.xAlrPrintHeadPsuFailure_B04');
	ELSIF EDGENEG(gInks[4].Al.xAlrPrintHeadPsuFailure) THEN
		MpAlarmXReset(gAlrCore, 'Inks.Alarm.inks.Al.xAlrPrintHeadPsuFailure_B04');
	END_IF

END_ACTION
```

### Program Logical/InkBox/Transport/Transport (IEC)

#### Transport.st
```iecst
PROGRAM _CYCLIC

	gToWriteDataModbTransport[1] := REAL_TO_UINT(gMachine.parSw.rBeltSpeedSetPoint*10);
	gToWriteDataModbTransport[2] := REAL_TO_UINT(gTransVacuum[1].parSw.rManSetPoint);
	gToWriteDataModbTransport[3] := REAL_TO_UINT(gBelt.parSw.rGearBox*10);
	gToWriteDataModbTransport[4] := REAL_TO_UINT(gBelt.parSw.rAxisLength);

	IF gInkBox.Commands.xReset THEN
		gToWriteDataModbTransport[5] := 1;
	ELSE
		gToWriteDataModbTransport[5] := 0;
	END_IF

	IF EDGEPOS(gBelt.commands.xRunBelt) THEN
		gToWriteDataModbTransport[6] := 1;
	ELSIF EDGENEG(gBelt.commands.xRunBelt) THEN
		gToWriteDataModbTransport[6] := 0;
	ELSIF gToWriteDataModbTransport[6] = 1 OR gToWriteDataModbTransport[6] = 0 THEN
		gToWriteDataModbTransport[6] := -1;
	END_IF

	IF EDGEPOS(gTransVacuum[1].OrdersSw.xRunManual) THEN
		gToWriteDataModbTransport[7] := 1;
	ELSIF EDGENEG(gTransVacuum[1].OrdersSw.xRunManual) THEN
		gToWriteDataModbTransport[7] := 0;
	ELSIF gToWriteDataModbTransport[7] = 1 OR gToWriteDataModbTransport[7] = 0 THEN
		gToWriteDataModbTransport[7] := -1;
	END_IF

	//Remove order of Belt when receiving a falling in the Status signal
	IF EDGEPOS(gReceivedDataModbTransport[5]=0 OR gReceivedDataModbTransport[5]=2) THEN
		gBelt.commands.xRunBelt := FALSE;
	END_IF

	//Remove order of Belt when receiving a falling in the Status signal
	IF EDGEPOS(gReceivedDataModbTransport[6]=0 OR gReceivedDataModbTransport[6]=2) THEN
		gTransVacuum[1].OrdersSw.xRunManual := FALSE;
	END_IF

	gBelt.Al.xAnyDriveAlarm := gReceivedDataModbTransport[5]=2;
	gTransVacuum[1].Alarms.xAlrBlowerError[1] := gReceivedDataModbTransport[6]=2;

END_PROGRAM
```

### AsARCfg.var
```iecst
VAR CONSTANT
	cfgERR_DEVICE_NOT_EXIST			: UINT		:= 29000;	(*device doesn't exist or device not configured*)
	cfgERR_DEVICE_INVALID			: UINT		:= 29001;	(*FBK "pDevice" parameter invalid (e.g. pDevice = 0)*)
	cfgERR_OPTION_INVALID			: UINT		:= 29002;	(*FBK "Option" parameter invalid*)
	cfgERR_VALUE_INVALID			: UINT		:= 29003;	(*invalid FBK parameter, error text depends on the function block*)
	cfgERR_SET_NOT_POSSIBLE			: UINT		:= 29004;	(*not possible to set the subnet mask (e.g. DHCP client)*)
	cfgERR_ARREG					: UINT		:= 29005;	(*error in the AR registry*)
	cfgERR_INANODE_NOT_SUPPORTED	: UINT		:= 29006;	(*INA device does not support INA node numbers (e.g. IF1 = RS232)*)
	cfgERR_FTP_SINIT				: UINT		:= 29007;	(*initialization error on FTP server*)
	cfgERR_FTP_SDOWN				: UINT		:= 29008;	(*shutdown error on FTP server*)
	cfgERR_PARAM_NOT_SET			: UINT		:= 29009;	(*default gateway not defined*)
	cfgERR_SNTP_SERVER 				: UINT		:= 29010;	(*could not start the SNTP server*)
	cfgERR_SNTP_CLIENT 				: UINT		:= 29011;	(*error starting SNTP client (e.g. client already running)*)
	cfgERR_SNTP_INTERVAL 			: UINT		:= 29012;	(*invalid FBK parameter - values from 1 to 60 are valid*)
	cfgERR_SYSTEM		 			: UINT		:= 29013;	(*unexpected system error*)
	cfgERR_TIMEZONE					: UINT		:= 29014;   (*invalid timezone specified*)
	cfgERR_YEAR_INVALID				: UINT		:= 29015;	(*invalid year specified*)
	cfgERR_CIFS_DOMAIN_INVALID		: UINT 		:= 29016;   (*cifs domain name not defined *)
	cfgERR_CIFS_DEFAULTUSER_INVALID	: UINT		:= 29017;	(*cifs defaultuser not defined *)
	cfgERR_INANODE_NUMBER_SET       : UINT      := 29018;	(*could not set the INA node number*)
	cfgERR_CIFS_DEFAULTPW_INVALID	: UINT		:= 29019;	(*cifs default password not defined *)
	cfgERR_DHCP_SERVER_STARTED		: UINT		:= 29020;	(*server is already working*)
	cfgERR_INTERFACELIST_BUFFER		: UINT		:= 29021;	(*interfacelist buffer to small*)
	cfgERR_LEASES_BUFFER			: UINT		:= 29022;	(*leases array to small*)
	cfgERR_LEASE_EXISTS				: UINT		:= 29023;	(*leasename already exists*)
	cfgERR_LEASE_TIMEOUT			: UINT		:= 29024;	(*invalid lease timeout*)
	cfgERR_DHCP_CONFIG				: UINT		:= 29025;	(*DHCP server is not configured*)
	cfgERR_SDM_FUNCTION_NOT_FOUND	: UINT		:= 29026;	(*used arsdm function was not found*)
	cfgERR_CLEAR_NV_DATA			: UINT		:= 29027;	(*could not clear NV data*)
	cfgERR_FUNCTION_NOT_FOUND	    : UINT		:= 29028;	(*referenced function was not found*)
	cfgERR_SDM_DISABLED 		    : UINT      := 29029;	(*System diagnostics disabled*)
	cfgERR_WEBSERV_DISABLED 		: UINT      := 29030;	(*Web Server disabled*)
	cfgERR_DHCP_NO_DHCP_IP_OBTAINED : UINT      := 29031;   (*DHCP activated, but no IP obtained*)
	cfgERR_NTP_SERVER 				: UINT		:= 29032;	(*could not start the NTP server*)
	cfgERR_NTP_CLIENT 				: UINT		:= 29033;	(*error starting NTP client*)
	cfgERR_ROUTE_TABLE				: UINT		:= 29034;	(*error updating network routing table*)

	cfgETHBAUDRATE_AUTO				: UDINT		:= 0;		(*auto-detect*)
	cfgETHBAUDRATE_10				: UDINT		:= 10;		(*10 MBaud, half-duplex*)
	cfgETHBAUDRATE_10FD				: UDINT		:= 11;		(*10 MBaud, full-duplex*)
	cfgETHBAUDRATE_100				: UDINT		:= 100;		(*100 MBaud, half-duplex*)
	cfgETHBAUDRATE_100FD			: UDINT		:= 101;		(*100 MBaud, full-duplex*)
	cfgETHBAUDRATE_1000FD			: UDINT		:= 1001;	(*1 GBaud, full-duplex*)

	cfgOPTION_NON_VOLATILE			: UDINT		:= 1;		(*permanently sets parameters*)
	cfgOPTION_VOLATILE				: UDINT		:= 0;		(*temporarily sets parameters*)

	cfgCONFIGMODE_MANUALLY			: UDINT		:= 0;		(*manual configuration*)
	cfgCONFIGMODE_DHCPCLIENT		: UDINT		:= 1;		(*DHCP client*)

	cfgOPTION_DISABLE				: UDINT		:= 0;		(*disable*)
	cfgOPTION_ENABLE				: UDINT		:= 1;		(*enable*)

	cfgOPTION_WORKGROUP				: USINT		:= 1;		(*Domain is Workgroup*)
	cfgOPTION_NON_WORKGROUP			: USINT		:= 0;		(*Domain isn't Workgroup*)

	cfgOPTION_ENABLE_SDM			: USINT		:= 1;		(*enable sdm*)
	cfgOPTION_DISABLE_SDM			: USINT		:= 2;		(*disable sdm*)

	cfgSTATUS_SDM_ENABLED			: USINT		:= 1;		(*sdm is enabled*)
	cfgSTATUS_SDM_DISABLED			: USINT		:= 2;		(*sdm is disabled*)

	cfgWEB_MODE_GOFORM_DISABLE		: UINT		:= 0;		(*Webserver Goform disabled*)
	cfgWEB_MODE_GOFORM_ENABLE		: UINT		:= 1;		(*Webserver Goform enabled*)
	cfgWEB_MODE_GOFORM_NO_WRITE		: UINT		:= 2;		(*Webserver Goform readonly*)

	cfgWEB_MODE_MIME_DEL			: UINT		:= 0;		(*Webserver delete MimeType*)
	cfgWEB_MODE_MIME_ADD			: UINT		:= 1;		(*Webserver set MimeType*)

	cfgWEB_MODE_DISABLED			: UINT		:= 0;		(*Webserver disabled*)
	cfgWEB_MODE_ENABLED				: UINT		:= 1;		(*Webserver enabled*)

	cfgOPTION_DNS_OFF				: USINT		:= 0;		(*disable DNS service*)
	cfgOPTION_DNS_ON_CONFIG			: USINT		:= 1;		(*DNS service using the server address as configured*)
	cfgOPTION_DNS_ON_DHCP			: USINT		:= 2;		(*Get the DNS address from the DHCP server*)

	cfgNTP_START					: UINT		:= 1;		(*start NTP server/client*)
	cfgNTP_STOP						: UINT		:= 0;		(*stop NTP server/client*)
	cfgSTATUS_NTP_ACTIVE			: UINT		:= 1;		(*NTP server/client active*)
	cfgSTATUS_NTP_INACTIVE			: UINT		:= 0;		(*NTP server/client inactive*)

	cfgSDM_COLOR_DEFAULT			: UDINT		:= 2147483648;	(*sdm default color*)

	cfgDHCP_OPTION_VENDOR_CLASS_ID	: USINT		:= 60; 		(*DHCP option vendor class identifier*)

END_VAR
```

### AsOpcUac.var
```iecst
VAR CONSTANT
	MAX_LENGTH_VARIABLE					: UINT := 255;
	MAX_LENGTH_BYTESTRING				: UINT := 1024;

	MAX_ELEMENTS_ARRAYDIMENSION 		: UINT := 7;	(* B&R supports arrays with 7 dimensions											*)
	MAX_ELEMENTS_INDEXRANGE 			: UINT := 8;	(* Index range addresses max number of dimensions +1 for string/bytestring index	*)
	MAX_ELEMENTS_NODELIST 				: UINT := 64;	(* Maximum number of items the node list functions can handle						*)
	MAX_ELEMENTS_MONITORLIST			: UINT := 64;	(* Maximum number of elements the monitored item list functions can handle			*)
	MAX_ELEMENTS_ARGUMENTS 				: UINT := 10;	(* Maximum number of input and output arguments for method call						*)
	MAX_ELEMENTS_EVENTFIELDSELECTION	: UINT := 64;
	MAX_ELEMENTS_RELATIVEPATH			: UINT := 16;

	(* B&R requires zero based arrays in .typ and .fun files, calculations like "const - 1" are not allowed
	   for declarations in those files, so other constants denoting the array upper limit are declared *)
	MAX_INDEX_ARRAYDIMENSION 			: UINT := MAX_ELEMENTS_ARRAYDIMENSION - 1;
	MAX_INDEX_INDEXRANGE 				: UINT := MAX_ELEMENTS_INDEXRANGE - 1;
	MAX_INDEX_NODELIST 					: UINT := MAX_ELEMENTS_NODELIST - 1;
	MAX_INDEX_MONITORLIST 				: UINT := MAX_ELEMENTS_MONITORLIST - 1;
	MAX_INDEX_ARGUMENTS 				: UINT := MAX_ELEMENTS_ARGUMENTS - 1;
	MAX_INDEX_EVENTFIELDSELECTION		: UINT := MAX_ELEMENTS_EVENTFIELDSELECTION - 1;
	MAX_INDEX_RELATIVEPATH				: UINT := MAX_ELEMENTS_RELATIVEPATH - 1;
	MAX_INDEX_BYTESTRING				: UINT := MAX_LENGTH_BYTESTRING - 1;
END_VAR
```

### Library Logical/Libraries/BRSE_JSON

#### BRSE_JSON.fun
```iecst
(********************************************************************
 * COPYRIGHT -- B&R
 ********************************************************************
 * Library: Library
 * File: Library.fun
 * Author: Florian Damerow
 * Created: March 09, 2011
 ********************************************************************
 * Functions and function blocks of library Library
 ********************************************************************)

FUNCTION_BLOCK JSON_Parse (*parses a JSON message and writes the content to the structure on the PLC*)
	VAR_INPUT
		pMessage : REFERENCE TO UDINT; (*Pointer to the JSON Message (String)*)
		pDebug : REFERENCE TO UDINT; (*Pointer Debug Buffer (String)*)
		pVariablesNotFound : REFERENCE TO UDINT; (*Pointer Buffer of VariablesNotFound (String)*)
		SizeVariablesNotFound : UDINT; (*size of the VariablesNotFound Buffer*)
		SizeDebug : UDINT; (*size of the Debug Buffer*)
		MaxLoopIdx : UDINT; (*Number of iterations per scan. Default 1000*)
	END_VAR
	VAR_OUTPUT
		ErrorInfo : UINT; (*Shows internal error messages*)
		Status : UINT; (*1: Done 2:Error*)
	END_VAR
	VAR
		parselevel : USINT;
		pvIndex : ARRAY[0..MAX_STRUCT_DEPTH_Parse] OF INT;
		Buffer : STRING[1000];
		parsestateold : USINT;
		parsestate : USINT;
		pvName : ARRAY[0..MAX_STRUCT_DEPTH_Parse] OF STRING[32];
		buffIdx : UDINT;
		isArray : ARRAY[0..MAX_STRUCT_DEPTH_Parse] OF BOOL;
		fullName : STRING[MAX_STRUCT_NAME_LENGTH_Parse];
		j : UINT;
		loopIdx : UDINT;
		messageLength : UDINT;
	END_VAR
END_FUNCTION_BLOCK

FUNCTION_BLOCK JSON_Stringify (*converts a PV variable and the whole structure into a JSON Object using PV_ninfo*)
	VAR_INPUT
		pStName : REFERENCE TO UDINT; (*address to variable name (STRING)*)
		MaxLoopIdx : UDINT; (*Number of iterations per scan. Default 1000*)
		pMessage : UDINT; (*Pointer to output buffer for the complete JSON string.*)
	END_VAR
	VAR_OUTPUT
		Status : UINT; (*address to status-variable 0=not done; 1=done; 2=error*)
		Output : STRING[MAX_OUTPUT_LENGTH_Stringify];
	END_VAR
	VAR
		tmpStruct : STRING[MAX_OUTPUT_LENGTH_Stringify];
		pvName : ARRAY[0..MAX_STRUCT_DEPTH_Stringify] OF STRING[100];
		j : UDINT;
		pvIndex : ARRAY[0..MAX_STRUCT_DEPTH_Stringify] OF UINT;
		TaskDoc : TaskDoc1_typ;
		pvType : UDINT;
		pvLength : UDINT;
		arrMem : ARRAY[0..MAX_STRUCT_DEPTH_Stringify] OF UINT;
		pvStructMembers : ARRAY[0..MAX_STRUCT_DEPTH_Stringify] OF UINT;
		tmpValue : STRING[MAX_OUTPUT_LENGTH_Stringify];
		Buffer : STRING[MAX_OUTPUT_LENGTH_Stringify];
		i : DINT;
		pvLevel : DINT;
		tmpDepth : STRING[MAX_OUTPUT_LENGTH_Stringify];
		state : USINT;
		pvContinue : BOOL;
		pvSearchComplete : BOOL;
		data_len : UDINT;
		isArray : ARRAY[0..MAX_STRUCT_DEPTH_Stringify] OF BOOL;
		arrIndex : USINT;
		pv_adresse : UDINT;
		loopIdx : UDINT;
		messageIdx : UDINT;
	END_VAR
END_FUNCTION_BLOCK
```

#### BRSE_JSON_Main.h
```c
/*! \file BRSE_JSON_Main.h */
/*!
	\mainpage BRSE_JSON

	\section Introduction
	\brief This library provides the ability to use JSON to write and read variables using normal ASCII string communication.

	This library can extract the members and their values within a structure variable into a JavaScriptObjectNotification string format,
	and parse the JSON-string back into a structure - eg. set the values of the structure members from the string information.

	See also <a href="http://www.json.org">http://www.json.org</a> for the JSON syntax.

	Useful for Javascript web pages or Java-written clients, or simply for storing structure data in a compact ASCII format.

	\section Usage
	The library contains two function blocks \ref JSON_Parse and \ref JSON_Stringify.

	\ref JSON_Parse takes a JSON string created by \ref JSON_Stringify and interprets it.
	It searches for the variables and updates their values on the PLC.

	\ref JSON_Stringify takes an address to a string containing a variable or structure name and creates a JSON string.
	The JSON string contains all the necessary data about the structure or variable so that a parser can reconstruct it.
	It uses a basic JSON structure: {name:content}

	An example of a string is the following:

	{"PV_var1":[{"Outer1":[{"Middle2":"1234","Middle1":[{"Inner1":"90","Inner2":"22","Inner3":"33"}]}]"Outer2":"567"}]}

	The JSON string describes the following structure:
	 	- PV_var1 \n
		- Outer1 \n
			- Middle2 1234 \n
			- Middle1 \n
				- Inner1 90 \n
				- Inner2 22 \n
				- Inner3 33 \n
		- Outer2 567

	\section Downloads
	There is an example package included.\n
	Please import into project via Add Existing Package.\n
	In the package there is an html javascript file. Please only run it in Internet Explorer. \n
	The example shows an basic "monitor" mode implementation using an webservice together with BRSE_JSON. \n
	<a href="y:\Application\Libraries\BRSE_JSON\Documentation\WEB_Interface.zip">WEB_interface</a><br><br>
	There is also a smaller test program just for testing the basic functionality.
	<a href="y:\Application\Libraries\BRSE_JSON\Documentation\TestProgram.zip">TestProgram</a><br><br>
	*/

#include "BRSE_JSON.h"
#include <string.h> /*this will override the asstring functions*/
```
